       // Index 0
       IF "HMI_Interface_Overview".homeCodition[8].pageIndex = 0 THEN
           "HMI_Interface_Overview".homeCodition[8].emOverviewTitle := WSTRING#'Home Condition 0';
           "HMI_Interface_Overview".homeCodition[8].emOverviewCmName[0] := WSTRING#'Thickness Z-Axis';
           "HMI_Interface_Overview".homeCodition[8].emOverviewCmName[1] := WSTRING#'Hipot & Thickness Servo Press';
           "HMI_Interface_Overview".homeCodition[8].emOverviewCmName[2] := WSTRING#'Hipot Tab Contactor Left';
           "HMI_Interface_Overview".homeCodition[8].emOverviewCmName[3] := WSTRING#'Hipot Tab Contactor Right';
           "HMI_Interface_Overview".homeCodition[8].emOverviewCmName[4] := WSTRING#'Hipot Tab Contactor';
           "HMI_Interface_Overview".homeCodition[8].emOverviewCmName[5] := WSTRING#'Hipot & Thickness Stage Lift Front';
           "HMI_Interface_Overview".homeCodition[8].emOverviewCmName[6] := WSTRING#'Hipot & Thickness Stage Lift Rear';
           "HMI_Interface_Overview".homeCodition[8].emOverviewCmName[7] := WSTRING#'Hipot & Thickness JR Detect';
           "HMI_Interface_Overview".homeCodition[8].emOverviewCmName[8] := WSTRING#'Spare';
           "HMI_Interface_Overview".homeCodition[8].emOverviewCmName[9] := WSTRING#'Spare';
           "HMI_Interface_Overview".homeCodition[8].emOverviewCmName[10] := WSTRING#'Spare';
           "HMI_Interface_Overview".homeCodition[8].emOverviewCmName[11] := WSTRING#'Spare';
           "HMI_Interface_Overview".homeCodition[8].emOverviewCmName[12] := WSTRING#'Spare';
           "HMI_Interface_Overview".homeCodition[8].emOverviewCmName[13] := WSTRING#'Spare';
           "HMI_Interface_Overview".homeCodition[8].emOverviewCmPositionName[0] := WSTRING#'Wait Position';
           "HMI_Interface_Overview".homeCodition[8].emOverviewCmPositionName[1] := WSTRING#'Home Position';
           "HMI_Interface_Overview".homeCodition[8].emOverviewCmPositionName[2] := WSTRING#'Open';
           "HMI_Interface_Overview".homeCodition[8].emOverviewCmPositionName[3] := WSTRING#'Open';
           "HMI_Interface_Overview".homeCodition[8].emOverviewCmPositionName[4] := WSTRING#'Backward';
           "HMI_Interface_Overview".homeCodition[8].emOverviewCmPositionName[5] := WSTRING#'Down';
           "HMI_Interface_Overview".homeCodition[8].emOverviewCmPositionName[6] := WSTRING#'Down';
           "HMI_Interface_Overview".homeCodition[8].emOverviewCmPositionName[7] := WSTRING#'Not Detect';
           "HMI_Interface_Overview".homeCodition[8].emOverviewCmPositionName[8] := WSTRING#'Spare';
           "HMI_Interface_Overview".homeCodition[8].emOverviewCmPositionName[9] := WSTRING#'Spare';
           "HMI_Interface_Overview".homeCodition[8].emOverviewCmPositionName[10] := WSTRING#'Spare';
           "HMI_Interface_Overview".homeCodition[8].emOverviewCmPositionName[11] := WSTRING#'Spare';
           "HMI_Interface_Overview".homeCodition[8].emOverviewCmPositionName[12] := WSTRING#'Spare';
           "HMI_Interface_Overview".homeCodition[8].emOverviewCmPositionName[13] := WSTRING#'Spare';
           IF NOT #statLampControl THEN
               "HMI_Interface_Overview".homeCodition[8].emOverviewHomeLampOn[0] := "Unit1.Em8.HmiInterface".cm.softcam.thicknessAxisZ.pos00_wait.inPos;
               "HMI_Interface_Overview".homeCodition[8].emOverviewHomeLampOn[1] := "Unit1.Em8.HmiInterface".cmHipotThicknessServoPress.monitoring.profinetInput."HOME-POS-REACHED";
               "HMI_Interface_Overview".homeCodition[8].emOverviewHomeLampOn[2] := "Unit1.Em8.HmiInterface".cmHipotTabContactorLeftOpenClose.monitoring.inHomePos;
               "HMI_Interface_Overview".homeCodition[8].emOverviewHomeLampOn[3] := "Unit1.Em8.HmiInterface".cmHipotTabContactorRightOpenClose.monitoring.inHomePos;
               "HMI_Interface_Overview".homeCodition[8].emOverviewHomeLampOn[4] := "Unit1.Em8.HmiInterface".cmHipotTabContactorBwdFwd.monitoring.inHomePos;
               "HMI_Interface_Overview".homeCodition[8].emOverviewHomeLampOn[5] := "Unit1.Em8.HmiInterface".cmHipotThicknessStageLiftFrontUpDown.monitoring.inWorkPos;
               "HMI_Interface_Overview".homeCodition[8].emOverviewHomeLampOn[6] := "Unit1.Em8.HmiInterface".cmHipotThicknessStageLiftRearUpDown.monitoring.inWorkPos;
               "HMI_Interface_Overview".homeCodition[8].emOverviewHomeLampOn[7] := NOT "Unit1.Em8.HmiInterface".cmHipotThicknessJRDetect.monitoring.processValue;
               "HMI_Interface_Overview".homeCodition[8].emOverviewHomeLampOn[8] := FALSE;
               "HMI_Interface_Overview".homeCodition[8].emOverviewHomeLampOn[9] := FALSE;
               "HMI_Interface_Overview".homeCodition[8].emOverviewHomeLampOn[10] := FALSE;
               "HMI_Interface_Overview".homeCodition[8].emOverviewHomeLampOn[11] := FALSE;
               "HMI_Interface_Overview".homeCodition[8].emOverviewHomeLampOn[12] := FALSE;
               "HMI_Interface_Overview".homeCodition[8].emOverviewHomeLampOn[13] := FALSE;
           END_IF;
       END_IF;

       // Index 1
       IF "HMI_Interface_Overview".homeCodition[8].pageIndex = 1 THEN
           "HMI_Interface_Overview".homeCodition[8].emOverviewTitle := WSTRING#'Home Condition 1';
           "HMI_Interface_Overview".homeCodition[8].emOverviewCmName[0] := WSTRING#'Thickness Z-Axis';
           "HMI_Interface_Overview".homeCodition[8].emOverviewCmName[1] := WSTRING#'Hipot & Thickness Servo Press';
           "HMI_Interface_Overview".homeCodition[8].emOverviewCmName[2] := WSTRING#'Hipot Tab Contactor Left';
           "HMI_Interface_Overview".homeCodition[8].emOverviewCmName[3] := WSTRING#'Hipot Tab Contactor Right';
           "HMI_Interface_Overview".homeCodition[8].emOverviewCmName[4] := WSTRING#'Hipot Tab Contactor';
           "HMI_Interface_Overview".homeCodition[8].emOverviewCmName[5] := WSTRING#'Hipot & Thickness Stage Lift Front';
           "HMI_Interface_Overview".homeCodition[8].emOverviewCmName[6] := WSTRING#'Hipot & Thickness Stage Lift Rear';
           "HMI_Interface_Overview".homeCodition[8].emOverviewCmName[7] := WSTRING#'Hipot & Thickness JR Detect';
           "HMI_Interface_Overview".homeCodition[8].emOverviewCmName[8] := WSTRING#'Spare';
           "HMI_Interface_Overview".homeCodition[8].emOverviewCmName[9] := WSTRING#'Spare';
           "HMI_Interface_Overview".homeCodition[8].emOverviewCmName[10] := WSTRING#'Spare';
           "HMI_Interface_Overview".homeCodition[8].emOverviewCmName[11] := WSTRING#'Spare';
           "HMI_Interface_Overview".homeCodition[8].emOverviewCmName[12] := WSTRING#'Spare';
           "HMI_Interface_Overview".homeCodition[8].emOverviewCmName[13] := WSTRING#'Spare';
           "HMI_Interface_Overview".homeCodition[8].emOverviewCmPositionName[0] := WSTRING#'Wait Position';
           "HMI_Interface_Overview".homeCodition[8].emOverviewCmPositionName[1] := WSTRING#'Home Position';
           "HMI_Interface_Overview".homeCodition[8].emOverviewCmPositionName[2] := WSTRING#'Open';
           "HMI_Interface_Overview".homeCodition[8].emOverviewCmPositionName[3] := WSTRING#'Open';
           "HMI_Interface_Overview".homeCodition[8].emOverviewCmPositionName[4] := WSTRING#'Backward';
           "HMI_Interface_Overview".homeCodition[8].emOverviewCmPositionName[5] := WSTRING#'Down';
           "HMI_Interface_Overview".homeCodition[8].emOverviewCmPositionName[6] := WSTRING#'Down';
           "HMI_Interface_Overview".homeCodition[8].emOverviewCmPositionName[7] := WSTRING#'Detect';
           "HMI_Interface_Overview".homeCodition[8].emOverviewCmPositionName[8] := WSTRING#'Spare';
           "HMI_Interface_Overview".homeCodition[8].emOverviewCmPositionName[9] := WSTRING#'Spare';
           "HMI_Interface_Overview".homeCodition[8].emOverviewCmPositionName[10] := WSTRING#'Spare';
           "HMI_Interface_Overview".homeCodition[8].emOverviewCmPositionName[11] := WSTRING#'Spare';
           "HMI_Interface_Overview".homeCodition[8].emOverviewCmPositionName[12] := WSTRING#'Spare';
           "HMI_Interface_Overview".homeCodition[8].emOverviewCmPositionName[13] := WSTRING#'Spare';
           IF NOT #statLampControl THEN
               "HMI_Interface_Overview".homeCodition[8].emOverviewHomeLampOn[0] := "Unit1.Em8.HmiInterface".cm.softcam.thicknessAxisZ.pos00_wait.inPos;
               "HMI_Interface_Overview".homeCodition[8].emOverviewHomeLampOn[1] := "Unit1.Em8.HmiInterface".cmHipotThicknessServoPress.monitoring.profinetInput."HOME-POS-REACHED";
               "HMI_Interface_Overview".homeCodition[8].emOverviewHomeLampOn[2] := "Unit1.Em8.HmiInterface".cmHipotTabContactorLeftOpenClose.monitoring.inHomePos;
               "HMI_Interface_Overview".homeCodition[8].emOverviewHomeLampOn[3] := "Unit1.Em8.HmiInterface".cmHipotTabContactorRightOpenClose.monitoring.inHomePos;
               "HMI_Interface_Overview".homeCodition[8].emOverviewHomeLampOn[4] := "Unit1.Em8.HmiInterface".cmHipotTabContactorBwdFwd.monitoring.inHomePos;
               "HMI_Interface_Overview".homeCodition[8].emOverviewHomeLampOn[5] := "Unit1.Em8.HmiInterface".cmHipotThicknessStageLiftFrontUpDown.monitoring.inWorkPos;
               "HMI_Interface_Overview".homeCodition[8].emOverviewHomeLampOn[6] := "Unit1.Em8.HmiInterface".cmHipotThicknessStageLiftRearUpDown.monitoring.inWorkPos;
               "HMI_Interface_Overview".homeCodition[8].emOverviewHomeLampOn[7] := "Unit1.Em8.HmiInterface".cmHipotThicknessJRDetect.monitoring.processValue;
               "HMI_Interface_Overview".homeCodition[8].emOverviewHomeLampOn[8] := FALSE;
               "HMI_Interface_Overview".homeCodition[8].emOverviewHomeLampOn[9] := FALSE;
               "HMI_Interface_Overview".homeCodition[8].emOverviewHomeLampOn[10] := FALSE;
               "HMI_Interface_Overview".homeCodition[8].emOverviewHomeLampOn[11] := FALSE;
               "HMI_Interface_Overview".homeCodition[8].emOverviewHomeLampOn[12] := FALSE;
               "HMI_Interface_Overview".homeCodition[8].emOverviewHomeLampOn[13] := FALSE;
           END_IF;
       END_IF;

   END_REGION
END_REGION

REGION Network 39 (SCL): Em 9 Page Index Mapping
   REGION Page Index

       // Index 0
       IF "HMI_Interface_Overview".homeCodition[9].pageIndex = 0 THEN
           "HMI_Interface_Overview".homeCodition[9].emOverviewTitle := WSTRING#'Home Condition 0';
           "HMI_Interface_Overview".homeCodition[9].emOverviewCmName[0] := WSTRING#'Vision Stage Lift';
           "HMI_Interface_Overview".homeCodition[9].emOverviewCmName[1] := WSTRING#'Vision Light';
           "HMI_Interface_Overview".homeCodition[9].emOverviewCmName[2] := WSTRING#'Vision JR Detect';
           "HMI_Interface_Overview".homeCodition[9].emOverviewCmName[3] := WSTRING#'Spare';
           "HMI_Interface_Overview".homeCodition[9].emOverviewCmName[4] := WSTRING#'Spare';
           "HMI_Interface_Overview".homeCodition[9].emOverviewCmName[5] := WSTRING#'Spare';
           "HMI_Interface_Overview".homeCodition[9].emOverviewCmName[6] := WSTRING#'Spare';
           "HMI_Interface_Overview".homeCodition[9].emOverviewCmName[7] := WSTRING#'Spare';
           "HMI_Interface_Overview".homeCodition[9].emOverviewCmName[8] := WSTRING#'Spare';
           "HMI_Interface_Overview".homeCodition[9].emOverviewCmName[9] := WSTRING#'Spare';
           "HMI_Interface_Overview".homeCodition[9].emOverviewCmName[10] := WSTRING#'Spare';
           "HMI_Interface_Overview".homeCodition[9].emOverviewCmName[11] := WSTRING#'Spare';
           "HMI_Interface_Overview".homeCodition[9].emOverviewCmName[12] := WSTRING#'Spare';
           "HMI_Interface_Overview".homeCodition[9].emOverviewCmName[13] := WSTRING#'Spare';
           "HMI_Interface_Overview".homeCodition[9].emOverviewCmPositionName[0] := WSTRING#'Down';
           "HMI_Interface_Overview".homeCodition[9].emOverviewCmPositionName[1] := WSTRING#'Up';
           "HMI_Interface_Overview".homeCodition[9].emOverviewCmPositionName[2] := WSTRING#'Not Detect';
           "HMI_Interface_Overview".homeCodition[9].emOverviewCmPositionName[3] := WSTRING#'Spare';
           "HMI_Interface_Overview".homeCodition[9].emOverviewCmPositionName[4] := WSTRING#'Spare';
           "HMI_Interface_Overview".homeCodition[9].emOverviewCmPositionName[5] := WSTRING#'Spare';
           "HMI_Interface_Overview".homeCodition[9].emOverviewCmPositionName[6] := WSTRING#'Spare';
           "HMI_Interface_Overview".homeCodition[9].emOverviewCmPositionName[7] := WSTRING#'Spare';
           "HMI_Interface_Overview".homeCodition[9].emOverviewCmPositionName[8] := WSTRING#'Spare';
           "HMI_Interface_Overview".homeCodition[9].emOverviewCmPositionName[9] := WSTRING#'Spare';
           "HMI_Interface_Overview".homeCodition[9].emOverviewCmPositionName[10] := WSTRING#'Spare';
           "HMI_Interface_Overview".homeCodition[9].emOverviewCmPositionName[11] := WSTRING#'Spare';
           "HMI_Interface_Overview".homeCodition[9].emOverviewCmPositionName[12] := WSTRING#'Spare';
           "HMI_Interface_Overview".homeCodition[9].emOverviewCmPositionName[13] := WSTRING#'Spare';
           IF NOT #statLampControl THEN
               "HMI_Interface_Overview".homeCodition[9].emOverviewHomeLampOn[0] := "Unit1.Em9.HmiInterface".cmVisionStageLiftUpDown.monitoring.inWorkPos;
               "HMI_Interface_Overview".homeCodition[9].emOverviewHomeLampOn[1] := "Unit1.Em9.HmiInterface".cmVisionLightUpDown.monitoring.inHomePos;
               "HMI_Interface_Overview".homeCodition[9].emOverviewHomeLampOn[2] := NOT "Unit1.Em9.HmiInterface".cmVisionJRDetect.monitoring.processValue;
               "HMI_Interface_Overview".homeCodition[9].emOverviewHomeLampOn[3] := FALSE;
               "HMI_Interface_Overview".homeCodition[9].emOverviewHomeLampOn[4] := FALSE;
               "HMI_Interface_Overview".homeCodition[9].emOverviewHomeLampOn[5] := FALSE;
               "HMI_Interface_Overview".homeCodition[9].emOverviewHomeLampOn[6] := FALSE;
               "HMI_Interface_Overview".homeCodition[9].emOverviewHomeLampOn[7] := FALSE;
               "HMI_Interface_Overview".homeCodition[9].emOverviewHomeLampOn[8] := FALSE;
               "HMI_Interface_Overview".homeCodition[9].emOverviewHomeLampOn[9] := FALSE;
               "HMI_Interface_Overview".homeCodition[9].emOverviewHomeLampOn[10] := FALSE;
               "HMI_Interface_Overview".homeCodition[9].emOverviewHomeLampOn[11] := FALSE;
               "HMI_Interface_Overview".homeCodition[9].emOverviewHomeLampOn[12] := FALSE;
               "HMI_Interface_Overview".homeCodition[9].emOverviewHomeLampOn[13] := FALSE;
           END_IF;
       END_IF;

       // Index 1
       IF "HMI_Interface_Overview".homeCodition[9].pageIndex = 1 THEN
           "HMI_Interface_Overview".homeCodition[9].emOverviewTitle := WSTRING#'Home Condition 1';
           "HMI_Interface_Overview".homeCodition[9].emOverviewCmName[0] := WSTRING#'Vision Stage Lift';
           "HMI_Interface_Overview".homeCodition[9].emOverviewCmName[1] := WSTRING#'Vision Light';
           "HMI_Interface_Overview".homeCodition[9].emOverviewCmName[2] := WSTRING#'Vision JR Detect';
           "HMI_Interface_Overview".homeCodition[9].emOverviewCmName[3] := WSTRING#'Spare';
           "HMI_Interface_Overview".homeCodition[9].emOverviewCmName[4] := WSTRING#'Spare';
           "HMI_Interface_Overview".homeCodition[9].emOverviewCmName[5] := WSTRING#'Spare';
           "HMI_Interface_Overview".homeCodition[9].emOverviewCmName[6] := WSTRING#'Spare';
           "HMI_Interface_Overview".homeCodition[9].emOverviewCmName[7] := WSTRING#'Spare';
           "HMI_Interface_Overview".homeCodition[9].emOverviewCmName[8] := WSTRING#'Spare';
           "HMI_Interface_Overview".homeCodition[9].emOverviewCmName[9] := WSTRING#'Spare';
           "HMI_Interface_Overview".homeCodition[9].emOverviewCmName[10] := WSTRING#'Spare';
           "HMI_Interface_Overview".homeCodition[9].emOverviewCmName[11] := WSTRING#'Spare';
           "HMI_Interface_Overview".homeCodition[9].emOverviewCmName[12] := WSTRING#'Spare';
           "HMI_Interface_Overview".homeCodition[9].emOverviewCmName[13] := WSTRING#'Spare';
           "HMI_Interface_Overview".homeCodition[9].emOverviewCmPositionName[0] := WSTRING#'Down';
           "HMI_Interface_Overview".homeCodition[9].emOverviewCmPositionName[1] := WSTRING#'Up';
           "HMI_Interface_Overview".homeCodition[9].emOverviewCmPositionName[2] := WSTRING#'Detect';
           "HMI_Interface_Overview".homeCodition[9].emOverviewCmPositionName[3] := WSTRING#'Spare';
           "HMI_Interface_Overview".homeCodition[9].emOverviewCmPositionName[4] := WSTRING#'Spare';
           "HMI_Interface_Overview".homeCodition[9].emOverviewCmPositionName[5] := WSTRING#'Spare';
           "HMI_Interface_Overview".homeCodition[9].emOverviewCmPositionName[6] := WSTRING#'Spare';
           "HMI_Interface_Overview".homeCodition[9].emOverviewCmPositionName[7] := WSTRING#'Spare';
           "HMI_Interface_Overview".homeCodition[9].emOverviewCmPositionName[8] := WSTRING#'Spare';
           "HMI_Interface_Overview".homeCodition[9].emOverviewCmPositionName[9] := WSTRING#'Spare';
           "HMI_Interface_Overview".homeCodition[9].emOverviewCmPositionName[10] := WSTRING#'Spare';
           "HMI_Interface_Overview".homeCodition[9].emOverviewCmPositionName[11] := WSTRING#'Spare';
           "HMI_Interface_Overview".homeCodition[9].emOverviewCmPositionName[12] := WSTRING#'Spare';
           "HMI_Interface_Overview".homeCodition[9].emOverviewCmPositionName[13] := WSTRING#'Spare';
           IF NOT #statLampControl THEN
               "HMI_Interface_Overview".homeCodition[9].emOverviewHomeLampOn[0] := "Unit1.Em9.HmiInterface".cmVisionStageLiftUpDown.monitoring.inWorkPos;
               "HMI_Interface_Overview".homeCodition[9].emOverviewHomeLampOn[1] := "Unit1.Em9.HmiInterface".cmVisionLightUpDown.monitoring.inHomePos;
               "HMI_Interface_Overview".homeCodition[9].emOverviewHomeLampOn[2] := "Unit1.Em9.HmiInterface".cmVisionJRDetect.monitoring.processValue;
               "HMI_Interface_Overview".homeCodition[9].emOverviewHomeLampOn[3] := FALSE;
               "HMI_Interface_Overview".homeCodition[9].emOverviewHomeLampOn[4] := FALSE;
               "HMI_Interface_Overview".homeCodition[9].emOverviewHomeLampOn[5] := FALSE;
               "HMI_Interface_Overview".homeCodition[9].emOverviewHomeLampOn[6] := FALSE;
               "HMI_Interface_Overview".homeCodition[9].emOverviewHomeLampOn[7] := FALSE;
               "HMI_Interface_Overview".homeCodition[9].emOverviewHomeLampOn[8] := FALSE;
               "HMI_Interface_Overview".homeCodition[9].emOverviewHomeLampOn[9] := FALSE;
               "HMI_Interface_Overview".homeCodition[9].emOverviewHomeLampOn[10] := FALSE;
               "HMI_Interface_Overview".homeCodition[9].emOverviewHomeLampOn[11] := FALSE;
               "HMI_Interface_Overview".homeCodition[9].emOverviewHomeLampOn[12] := FALSE;
               "HMI_Interface_Overview".homeCodition[9].emOverviewHomeLampOn[13] := FALSE;
           END_IF;
       END_IF;

   END_REGION
END_REGION

REGION Network 40 (SCL): Em 10 Page Index Mapping
   REGION Page Index

       // Index 0
       IF "HMI_Interface_Overview".homeCodition[10].pageIndex = 0 THEN
           "HMI_Interface_Overview".homeCodition[10].emOverviewTitle := WSTRING#'Home Condition 0';
           "HMI_Interface_Overview".homeCodition[10].emOverviewCmName[0] := WSTRING#'Laser Mark Stage Lift';
           "HMI_Interface_Overview".homeCodition[10].emOverviewCmName[1] := WSTRING#'Laser Mark Cover';
           "HMI_Interface_Overview".homeCodition[10].emOverviewCmName[2] := WSTRING#'Laser Mark JR Detect';
           "HMI_Interface_Overview".homeCodition[10].emOverviewCmName[3] := WSTRING#'Spare';
           "HMI_Interface_Overview".homeCodition[10].emOverviewCmName[4] := WSTRING#'Spare';
           "HMI_Interface_Overview".homeCodition[10].emOverviewCmName[5] := WSTRING#'Spare';
           "HMI_Interface_Overview".homeCodition[10].emOverviewCmName[6] := WSTRING#'Spare';
           "HMI_Interface_Overview".homeCodition[10].emOverviewCmName[7] := WSTRING#'Spare';
           "HMI_Interface_Overview".homeCodition[10].emOverviewCmName[8] := WSTRING#'Spare';
           "HMI_Interface_Overview".homeCodition[10].emOverviewCmName[9] := WSTRING#'Spare';
           "HMI_Interface_Overview".homeCodition[10].emOverviewCmName[10] := WSTRING#'Spare';
           "HMI_Interface_Overview".homeCodition[10].emOverviewCmName[11] := WSTRING#'Spare';
           "HMI_Interface_Overview".homeCodition[10].emOverviewCmName[12] := WSTRING#'Spare';
           "HMI_Interface_Overview".homeCodition[10].emOverviewCmName[13] := WSTRING#'Spare';
           "HMI_Interface_Overview".homeCodition[10].emOverviewCmPositionName[0] := WSTRING#'Down';
           "HMI_Interface_Overview".homeCodition[10].emOverviewCmPositionName[1] := WSTRING#'Up';
           "HMI_Interface_Overview".homeCodition[10].emOverviewCmPositionName[2] := WSTRING#'Not Detect';
           "HMI_Interface_Overview".homeCodition[10].emOverviewCmPositionName[3] := WSTRING#'Spare';
           "HMI_Interface_Overview".homeCodition[10].emOverviewCmPositionName[4] := WSTRING#'Spare';
           "HMI_Interface_Overview".homeCodition[10].emOverviewCmPositionName[5] := WSTRING#'Spare';
           "HMI_Interface_Overview".homeCodition[10].emOverviewCmPositionName[6] := WSTRING#'Spare';
           "HMI_Interface_Overview".homeCodition[10].emOverviewCmPositionName[7] := WSTRING#'Spare';
           "HMI_Interface_Overview".homeCodition[10].emOverviewCmPositionName[8] := WSTRING#'Spare';
           "HMI_Interface_Overview".homeCodition[10].emOverviewCmPositionName[9] := WSTRING#'Spare';
           "HMI_Interface_Overview".homeCodition[10].emOverviewCmPositionName[10] := WSTRING#'Spare';
           "HMI_Interface_Overview".homeCodition[10].emOverviewCmPositionName[11] := WSTRING#'Spare';
           "HMI_Interface_Overview".homeCodition[10].emOverviewCmPositionName[12] := WSTRING#'Spare';
           "HMI_Interface_Overview".homeCodition[10].emOverviewCmPositionName[13] := WSTRING#'Spare';
           IF NOT #statLampControl THEN
               "HMI_Interface_Overview".homeCodition[10].emOverviewHomeLampOn[0] := "Unit1.Em10.HmiInterface".cmLaserMarkStageLiftUpDown.monitoring.inWorkPos;
               "HMI_Interface_Overview".homeCodition[10].emOverviewHomeLampOn[1] := "Unit1.Em10.HmiInterface".cmLaserMarkCoverUpDown.monitoring.inHomePos;
               "HMI_Interface_Overview".homeCodition[10].emOverviewHomeLampOn[2] := NOT "Unit1.Em10.HmiInterface".cmLaserMarkJRDetect.monitoring.processValue;
               "HMI_Interface_Overview".homeCodition[10].emOverviewHomeLampOn[3] := FALSE;
               "HMI_Interface_Overview".homeCodition[10].emOverviewHomeLampOn[4] := FALSE;
               "HMI_Interface_Overview".homeCodition[10].emOverviewHomeLampOn[5] := FALSE;
               "HMI_Interface_Overview".homeCodition[10].emOverviewHomeLampOn[6] := FALSE;
               "HMI_Interface_Overview".homeCodition[10].emOverviewHomeLampOn[7] := FALSE;
               "HMI_Interface_Overview".homeCodition[10].emOverviewHomeLampOn[8] := FALSE;
               "HMI_Interface_Overview".homeCodition[10].emOverviewHomeLampOn[9] := FALSE;
               "HMI_Interface_Overview".homeCodition[10].emOverviewHomeLampOn[10] := FALSE;
               "HMI_Interface_Overview".homeCodition[10].emOverviewHomeLampOn[11] := FALSE;
               "HMI_Interface_Overview".homeCodition[10].emOverviewHomeLampOn[12] := FALSE;
               "HMI_Interface_Overview".homeCodition[10].emOverviewHomeLampOn[13] := FALSE;
           END_IF;
       END_IF;

       // Index 1
       IF "HMI_Interface_Overview".homeCodition[10].pageIndex = 1 THEN
           "HMI_Interface_Overview".homeCodition[10].emOverviewTitle := WSTRING#'Home Condition 1';
           "HMI_Interface_Overview".homeCodition[10].emOverviewCmName[0] := WSTRING#'Laser Mark Stage Lift';
           "HMI_Interface_Overview".homeCodition[10].emOverviewCmName[1] := WSTRING#'Laser Mark Cover';
           "HMI_Interface_Overview".homeCodition[10].emOverviewCmName[2] := WSTRING#'Laser Mark JR Detect';
           "HMI_Interface_Overview".homeCodition[10].emOverviewCmName[3] := WSTRING#'Spare';
           "HMI_Interface_Overview".homeCodition[10].emOverviewCmName[4] := WSTRING#'Spare';
           "HMI_Interface_Overview".homeCodition[10].emOverviewCmName[5] := WSTRING#'Spare';
           "HMI_Interface_Overview".homeCodition[10].emOverviewCmName[6] := WSTRING#'Spare';
           "HMI_Interface_Overview".homeCodition[10].emOverviewCmName[7] := WSTRING#'Spare';
           "HMI_Interface_Overview".homeCodition[10].emOverviewCmName[8] := WSTRING#'Spare';
           "HMI_Interface_Overview".homeCodition[10].emOverviewCmName[9] := WSTRING#'Spare';
           "HMI_Interface_Overview".homeCodition[10].emOverviewCmName[10] := WSTRING#'Spare';
           "HMI_Interface_Overview".homeCodition[10].emOverviewCmName[11] := WSTRING#'Spare';
           "HMI_Interface_Overview".homeCodition[10].emOverviewCmName[12] := WSTRING#'Spare';
           "HMI_Interface_Overview".homeCodition[10].emOverviewCmName[13] := WSTRING#'Spare';
           "HMI_Interface_Overview".homeCodition[10].emOverviewCmPositionName[0] := WSTRING#'Down';
           "HMI_Interface_Overview".homeCodition[10].emOverviewCmPositionName[1] := WSTRING#'Up';
           "HMI_Interface_Overview".homeCodition[10].emOverviewCmPositionName[2] := WSTRING#'Detect';
           "HMI_Interface_Overview".homeCodition[10].emOverviewCmPositionName[3] := WSTRING#'Spare';
           "HMI_Interface_Overview".homeCodition[10].emOverviewCmPositionName[4] := WSTRING#'Spare';
           "HMI_Interface_Overview".homeCodition[10].emOverviewCmPositionName[5] := WSTRING#'Spare';
           "HMI_Interface_Overview".homeCodition[10].emOverviewCmPositionName[6] := WSTRING#'Spare';
           "HMI_Interface_Overview".homeCodition[10].emOverviewCmPositionName[7] := WSTRING#'Spare';
           "HMI_Interface_Overview".homeCodition[10].emOverviewCmPositionName[8] := WSTRING#'Spare';
           "HMI_Interface_Overview".homeCodition[10].emOverviewCmPositionName[9] := WSTRING#'Spare';
           "HMI_Interface_Overview".homeCodition[10].emOverviewCmPositionName[10] := WSTRING#'Spare';
           "HMI_Interface_Overview".homeCodition[10].emOverviewCmPositionName[11] := WSTRING#'Spare';
           "HMI_Interface_Overview".homeCodition[10].emOverviewCmPositionName[12] := WSTRING#'Spare';
           "HMI_Interface_Overview".homeCodition[10].emOverviewCmPositionName[13] := WSTRING#'Spare';
           IF NOT #statLampControl THEN
               "HMI_Interface_Overview".homeCodition[10].emOverviewHomeLampOn[0] := "Unit1.Em10.HmiInterface".cmLaserMarkStageLiftUpDown.monitoring.inWorkPos;
               "HMI_Interface_Overview".homeCodition[10].emOverviewHomeLampOn[1] := "Unit1.Em10.HmiInterface".cmLaserMarkCoverUpDown.monitoring.inHomePos;
               "HMI_Interface_Overview".homeCodition[10].emOverviewHomeLampOn[2] := "Unit1.Em10.HmiInterface".cmLaserMarkJRDetect.monitoring.processValue;
               "HMI_Interface_Overview".homeCodition[10].emOverviewHomeLampOn[3] := FALSE;
               "HMI_Interface_Overview".homeCodition[10].emOverviewHomeLampOn[4] := FALSE;
               "HMI_Interface_Overview".homeCodition[10].emOverviewHomeLampOn[5] := FALSE;
               "HMI_Interface_Overview".homeCodition[10].emOverviewHomeLampOn[6] := FALSE;
               "HMI_Interface_Overview".homeCodition[10].emOverviewHomeLampOn[7] := FALSE;
               "HMI_Interface_Overview".homeCodition[10].emOverviewHomeLampOn[8] := FALSE;
               "HMI_Interface_Overview".homeCodition[10].emOverviewHomeLampOn[9] := FALSE;
               "HMI_Interface_Overview".homeCodition[10].emOverviewHomeLampOn[10] := FALSE;
               "HMI_Interface_Overview".homeCodition[10].emOverviewHomeLampOn[11] := FALSE;
               "HMI_Interface_Overview".homeCodition[10].emOverviewHomeLampOn[12] := FALSE;
               "HMI_Interface_Overview".homeCodition[10].emOverviewHomeLampOn[13] := FALSE;
           END_IF;
       END_IF;

   END_REGION
END_REGION

REGION Network 41 (SCL): Em 12 Page Index Mapping
   REGION Page Index

       // Index 0
       IF "HMI_Interface_Overview".homeCodition[12].pageIndex = 0 THEN
           "HMI_Interface_Overview".homeCodition[12].emOverviewTitle := WSTRING#'Home Condition 0';
           "HMI_Interface_Overview".homeCodition[12].emOverviewCmName[0] := WSTRING#'Stack NG Box Loading';
           "HMI_Interface_Overview".homeCodition[12].emOverviewCmName[1] := WSTRING#'Stack NG Box Unit Mover';
           "HMI_Interface_Overview".homeCodition[12].emOverviewCmName[2] := WSTRING#'Stack NG Box Clamp Left ';
           "HMI_Interface_Overview".homeCodition[12].emOverviewCmName[3] := WSTRING#'Stack NG Box Clamp Right';
           "HMI_Interface_Overview".homeCodition[12].emOverviewCmName[4] := WSTRING#'Stack NG Box Clamp Mover';
           "HMI_Interface_Overview".homeCodition[12].emOverviewCmName[5] := WSTRING#'Spare';
           "HMI_Interface_Overview".homeCodition[12].emOverviewCmName[6] := WSTRING#'Spare';
           "HMI_Interface_Overview".homeCodition[12].emOverviewCmName[7] := WSTRING#'Spare';
           "HMI_Interface_Overview".homeCodition[12].emOverviewCmName[8] := WSTRING#'Spare';
           "HMI_Interface_Overview".homeCodition[12].emOverviewCmName[9] := WSTRING#'Spare';
           "HMI_Interface_Overview".homeCodition[12].emOverviewCmName[10] := WSTRING#'Spare';
           "HMI_Interface_Overview".homeCodition[12].emOverviewCmName[11] := WSTRING#'Spare';
           "HMI_Interface_Overview".homeCodition[12].emOverviewCmName[12] := WSTRING#'Spare';
           "HMI_Interface_Overview".homeCodition[12].emOverviewCmName[13] := WSTRING#'Spare';
           "HMI_Interface_Overview".homeCodition[12].emOverviewCmPositionName[0] := WSTRING#'Up';
           "HMI_Interface_Overview".homeCodition[12].emOverviewCmPositionName[1] := WSTRING#'Forward';
           "HMI_Interface_Overview".homeCodition[12].emOverviewCmPositionName[2] := WSTRING#'Open';
           "HMI_Interface_Overview".homeCodition[12].emOverviewCmPositionName[3] := WSTRING#'Open';
           "HMI_Interface_Overview".homeCodition[12].emOverviewCmPositionName[4] := WSTRING#'Open';
           "HMI_Interface_Overview".homeCodition[12].emOverviewCmPositionName[5] := WSTRING#'Spare';
           "HMI_Interface_Overview".homeCodition[12].emOverviewCmPositionName[6] := WSTRING#'Spare';
           "HMI_Interface_Overview".homeCodition[12].emOverviewCmPositionName[7] := WSTRING#'Spare';
           "HMI_Interface_Overview".homeCodition[12].emOverviewCmPositionName[8] := WSTRING#'Spare';
           "HMI_Interface_Overview".homeCodition[12].emOverviewCmPositionName[9] := WSTRING#'Spare';
           "HMI_Interface_Overview".homeCodition[12].emOverviewCmPositionName[10] := WSTRING#'Spare';
           "HMI_Interface_Overview".homeCodition[12].emOverviewCmPositionName[11] := WSTRING#'Spare';
           "HMI_Interface_Overview".homeCodition[12].emOverviewCmPositionName[12] := WSTRING#'Spare';
           "HMI_Interface_Overview".homeCodition[12].emOverviewCmPositionName[13] := WSTRING#'Spare';
           IF NOT #statLampControl THEN
               "HMI_Interface_Overview".homeCodition[12].emOverviewHomeLampOn[0] := "Unit1.Em12.HmiInterface".cmStackNgBoxLoadingUpDown.monitoring.inHomePos;
               "HMI_Interface_Overview".homeCodition[12].emOverviewHomeLampOn[1] := "Unit1.Em12.HmiInterface".cmStackNgBoxUnitMoverBwdFwd.monitoring.inWorkPos;
               "HMI_Interface_Overview".homeCodition[12].emOverviewHomeLampOn[2] := "Unit1.Em12.HmiInterface".cmStackNgBoxClampLeftOpenClose.monitoring.inHomePos;
               "HMI_Interface_Overview".homeCodition[12].emOverviewHomeLampOn[3] := "Unit1.Em12.HmiInterface".cmStackNgBoxClampRightOpenClose.monitoring.inHomePos;
               "HMI_Interface_Overview".homeCodition[12].emOverviewHomeLampOn[4] := "Unit1.Em12.HmiInterface".cmStackNgBoxClampMoverOpenClose.monitoring.inHomePos;
               "HMI_Interface_Overview".homeCodition[12].emOverviewHomeLampOn[5] := FALSE;
               "HMI_Interface_Overview".homeCodition[12].emOverviewHomeLampOn[6] := FALSE;
               "HMI_Interface_Overview".homeCodition[12].emOverviewHomeLampOn[7] := FALSE;
               "HMI_Interface_Overview".homeCodition[12].emOverviewHomeLampOn[8] := FALSE;
               "HMI_Interface_Overview".homeCodition[12].emOverviewHomeLampOn[9] := FALSE;
               "HMI_Interface_Overview".homeCodition[12].emOverviewHomeLampOn[10] := FALSE;
               "HMI_Interface_Overview".homeCodition[12].emOverviewHomeLampOn[11] := FALSE;
               "HMI_Interface_Overview".homeCodition[12].emOverviewHomeLampOn[12] := FALSE;
               "HMI_Interface_Overview".homeCodition[12].emOverviewHomeLampOn[13] := FALSE;
           END_IF;
       END_IF;

       // Index 1
       IF "HMI_Interface_Overview".homeCodition[12].pageIndex = 1 THEN
           "HMI_Interface_Overview".homeCodition[12].emOverviewTitle := WSTRING#'Home Condition 1';
           "HMI_Interface_Overview".homeCodition[12].emOverviewCmName[0] := WSTRING#'Stack NG Box Loading';
           "HMI_Interface_Overview".homeCodition[12].emOverviewCmName[1] := WSTRING#'Stack NG Box Unit Mover';
           "HMI_Interface_Overview".homeCodition[12].emOverviewCmName[2] := WSTRING#'Stack NG Box Clamp Left ';
           "HMI_Interface_Overview".homeCodition[12].emOverviewCmName[3] := WSTRING#'Stack NG Box Clamp Right';
           "HMI_Interface_Overview".homeCodition[12].emOverviewCmName[4] := WSTRING#'Stack NG Box Clamp Mover';
           "HMI_Interface_Overview".homeCodition[12].emOverviewCmName[5] := WSTRING#'Spare';
           "HMI_Interface_Overview".homeCodition[12].emOverviewCmName[6] := WSTRING#'Spare';
           "HMI_Interface_Overview".homeCodition[12].emOverviewCmName[7] := WSTRING#'Spare';
           "HMI_Interface_Overview".homeCodition[12].emOverviewCmName[8] := WSTRING#'Spare';
           "HMI_Interface_Overview".homeCodition[12].emOverviewCmName[9] := WSTRING#'Spare';
           "HMI_Interface_Overview".homeCodition[12].emOverviewCmName[10] := WSTRING#'Spare';
           "HMI_Interface_Overview".homeCodition[12].emOverviewCmName[11] := WSTRING#'Spare';
           "HMI_Interface_Overview".homeCodition[12].emOverviewCmName[12] := WSTRING#'Spare';
           "HMI_Interface_Overview".homeCodition[12].emOverviewCmName[13] := WSTRING#'Spare';
           "HMI_Interface_Overview".homeCodition[12].emOverviewCmPositionName[0] := WSTRING#'Up';
           "HMI_Interface_Overview".homeCodition[12].emOverviewCmPositionName[1] := WSTRING#'Forward';
           "HMI_Interface_Overview".homeCodition[12].emOverviewCmPositionName[2] := WSTRING#'Close';
           "HMI_Interface_Overview".homeCodition[12].emOverviewCmPositionName[3] := WSTRING#'Close';
           "HMI_Interface_Overview".homeCodition[12].emOverviewCmPositionName[4] := WSTRING#'Close';
           "HMI_Interface_Overview".homeCodition[12].emOverviewCmPositionName[5] := WSTRING#'Spare';
           "HMI_Interface_Overview".homeCodition[12].emOverviewCmPositionName[6] := WSTRING#'Spare';
           "HMI_Interface_Overview".homeCodition[12].emOverviewCmPositionName[7] := WSTRING#'Spare';
           "HMI_Interface_Overview".homeCodition[12].emOverviewCmPositionName[8] := WSTRING#'Spare';
           "HMI_Interface_Overview".homeCodition[12].emOverviewCmPositionName[9] := WSTRING#'Spare';
           "HMI_Interface_Overview".homeCodition[12].emOverviewCmPositionName[10] := WSTRING#'Spare';
           "HMI_Interface_Overview".homeCodition[12].emOverviewCmPositionName[11] := WSTRING#'Spare';
           "HMI_Interface_Overview".homeCodition[12].emOverviewCmPositionName[12] := WSTRING#'Spare';
           "HMI_Interface_Overview".homeCodition[12].emOverviewCmPositionName[13] := WSTRING#'Spare';
           IF NOT #statLampControl THEN
               "HMI_Interface_Overview".homeCodition[12].emOverviewHomeLampOn[0] := "Unit1.Em12.HmiInterface".cmStackNgBoxLoadingUpDown.monitoring.inHomePos;
               "HMI_Interface_Overview".homeCodition[12].emOverviewHomeLampOn[1] := "Unit1.Em12.HmiInterface".cmStackNgBoxUnitMoverBwdFwd.monitoring.inWorkPos;
               "HMI_Interface_Overview".homeCodition[12].emOverviewHomeLampOn[2] := "Unit1.Em12.HmiInterface".cmStackNgBoxClampLeftOpenClose.monitoring.inWorkPos;
               "HMI_Interface_Overview".homeCodition[12].emOverviewHomeLampOn[3] := "Unit1.Em12.HmiInterface".cmStackNgBoxClampRightOpenClose.monitoring.inWorkPos;
               "HMI_Interface_Overview".homeCodition[12].emOverviewHomeLampOn[4] := "Unit1.Em12.HmiInterface".cmStackNgBoxClampMoverOpenClose.monitoring.inWorkPos;
               "HMI_Interface_Overview".homeCodition[12].emOverviewHomeLampOn[5] := FALSE;
               "HMI_Interface_Overview".homeCodition[12].emOverviewHomeLampOn[6] := FALSE;
               "HMI_Interface_Overview".homeCodition[12].emOverviewHomeLampOn[7] := FALSE;
               "HMI_Interface_Overview".homeCodition[12].emOverviewHomeLampOn[8] := FALSE;
               "HMI_Interface_Overview".homeCodition[12].emOverviewHomeLampOn[9] := FALSE;
               "HMI_Interface_Overview".homeCodition[12].emOverviewHomeLampOn[10] := FALSE;
               "HMI_Interface_Overview".homeCodition[12].emOverviewHomeLampOn[11] := FALSE;
               "HMI_Interface_Overview".homeCodition[12].emOverviewHomeLampOn[12] := FALSE;
               "HMI_Interface_Overview".homeCodition[12].emOverviewHomeLampOn[13] := FALSE;
           END_IF;
       END_IF;

   END_REGION
END_REGION

REGION Network 42 (SCL): Em 13 Page Index Mapping
   REGION Page Index

       // Index 0
       IF "HMI_Interface_Overview".homeCodition[13].pageIndex = 0 THEN
           "HMI_Interface_Overview".homeCodition[13].emOverviewTitle := WSTRING#'Home Condition 0';
           "HMI_Interface_Overview".homeCodition[13].emOverviewCmName[0] := WSTRING#'JR Unloading P&P X-Axis';
           "HMI_Interface_Overview".homeCodition[13].emOverviewCmName[1] := WSTRING#'JR Unloading P&P Z-Axis';
           "HMI_Interface_Overview".homeCodition[13].emOverviewCmName[2] := WSTRING#'JR Unloading P&P C-Axis';
           "HMI_Interface_Overview".homeCodition[13].emOverviewCmName[3] := WSTRING#'JR Unloading P&P Clamp';
           "HMI_Interface_Overview".homeCodition[13].emOverviewCmName[4] := WSTRING#'JR Unloading P&P JR Detect';
           "HMI_Interface_Overview".homeCodition[13].emOverviewCmName[5] := WSTRING#'Spare';
           "HMI_Interface_Overview".homeCodition[13].emOverviewCmName[6] := WSTRING#'Spare';
           "HMI_Interface_Overview".homeCodition[13].emOverviewCmName[7] := WSTRING#'Spare';
           "HMI_Interface_Overview".homeCodition[13].emOverviewCmName[8] := WSTRING#'Spare';
           "HMI_Interface_Overview".homeCodition[13].emOverviewCmName[9] := WSTRING#'Spare';
           "HMI_Interface_Overview".homeCodition[13].emOverviewCmName[10] := WSTRING#'Spare';
           "HMI_Interface_Overview".homeCodition[13].emOverviewCmName[11] := WSTRING#'Spare';
           "HMI_Interface_Overview".homeCodition[13].emOverviewCmName[12] := WSTRING#'Spare';
           "HMI_Interface_Overview".homeCodition[13].emOverviewCmName[13] := WSTRING#'Spare';
           "HMI_Interface_Overview".homeCodition[13].emOverviewCmPositionName[0] := WSTRING#'Wait Position';
           "HMI_Interface_Overview".homeCodition[13].emOverviewCmPositionName[1] := WSTRING#'Wait Position';
           "HMI_Interface_Overview".homeCodition[13].emOverviewCmPositionName[2] := WSTRING#'Wait Position';
           "HMI_Interface_Overview".homeCodition[13].emOverviewCmPositionName[3] := WSTRING#'Open';
           "HMI_Interface_Overview".homeCodition[13].emOverviewCmPositionName[4] := WSTRING#'Not Detect';
           "HMI_Interface_Overview".homeCodition[13].emOverviewCmPositionName[5] := WSTRING#'Spare';
           "HMI_Interface_Overview".homeCodition[13].emOverviewCmPositionName[6] := WSTRING#'Spare';
           "HMI_Interface_Overview".homeCodition[13].emOverviewCmPositionName[7] := WSTRING#'Spare';
           "HMI_Interface_Overview".homeCodition[13].emOverviewCmPositionName[8] := WSTRING#'Spare';
           "HMI_Interface_Overview".homeCodition[13].emOverviewCmPositionName[9] := WSTRING#'Spare';
           "HMI_Interface_Overview".homeCodition[13].emOverviewCmPositionName[10] := WSTRING#'Spare';
           "HMI_Interface_Overview".homeCodition[13].emOverviewCmPositionName[11] := WSTRING#'Spare';
           "HMI_Interface_Overview".homeCodition[13].emOverviewCmPositionName[12] := WSTRING#'Spare';
           "HMI_Interface_Overview".homeCodition[13].emOverviewCmPositionName[13] := WSTRING#'Spare';
           IF NOT #statLampControl THEN
               "HMI_Interface_Overview".homeCodition[13].emOverviewHomeLampOn[0] := "Unit1.Em13.HmiInterface".cm.softcam.jrUnIoadingPnPAxisX.pos00_wait.inPos;
               "HMI_Interface_Overview".homeCodition[13].emOverviewHomeLampOn[1] := "Unit1.Em13.HmiInterface".cm.softcam.jrUnIoadingPnPAxisZ.pos00_wait.inPos;
               "HMI_Interface_Overview".homeCodition[13].emOverviewHomeLampOn[2] := "Unit1.Em13.HmiInterface".cm.softcam.jrUnIoadingPnPAxisC.pos00_wait.inPos;
               "HMI_Interface_Overview".homeCodition[13].emOverviewHomeLampOn[3] := "Unit1.Em13.HmiInterface".cmJRUnloadingPnPClampOpenClose.monitoring.inHomePos;
               "HMI_Interface_Overview".homeCodition[13].emOverviewHomeLampOn[4] := NOT "Unit1.Em13.HmiInterface".cmJRUnloadingPnPJRDetect.monitoring.processValue;
               "HMI_Interface_Overview".homeCodition[13].emOverviewHomeLampOn[5] := FALSE;
               "HMI_Interface_Overview".homeCodition[13].emOverviewHomeLampOn[6] := FALSE;
               "HMI_Interface_Overview".homeCodition[13].emOverviewHomeLampOn[7] := FALSE;
               "HMI_Interface_Overview".homeCodition[13].emOverviewHomeLampOn[8] := FALSE;
               "HMI_Interface_Overview".homeCodition[13].emOverviewHomeLampOn[9] := FALSE;
               "HMI_Interface_Overview".homeCodition[13].emOverviewHomeLampOn[10] := FALSE;
               "HMI_Interface_Overview".homeCodition[13].emOverviewHomeLampOn[11] := FALSE;
               "HMI_Interface_Overview".homeCodition[13].emOverviewHomeLampOn[12] := FALSE;
               "HMI_Interface_Overview".homeCodition[13].emOverviewHomeLampOn[13] := FALSE;
           END_IF;
       END_IF;

       // Index 1
       IF "HMI_Interface_Overview".homeCodition[13].pageIndex = 1 THEN
           "HMI_Interface_Overview".homeCodition[13].emOverviewTitle := WSTRING#'Home Condition 1';
           "HMI_Interface_Overview".homeCodition[13].emOverviewCmName[0] := WSTRING#'JR Unloading P&P X-Axis';
           "HMI_Interface_Overview".homeCodition[13].emOverviewCmName[1] := WSTRING#'JR Unloading P&P Z-Axis';
           "HMI_Interface_Overview".homeCodition[13].emOverviewCmName[2] := WSTRING#'JR Unloading P&P C-Axis';
           "HMI_Interface_Overview".homeCodition[13].emOverviewCmName[3] := WSTRING#'JR Unloading P&P Clamp';
           "HMI_Interface_Overview".homeCodition[13].emOverviewCmName[4] := WSTRING#'JR Unloading P&P JR Detect';
           "HMI_Interface_Overview".homeCodition[13].emOverviewCmName[5] := WSTRING#'Spare';
           "HMI_Interface_Overview".homeCodition[13].emOverviewCmName[6] := WSTRING#'Spare';
           "HMI_Interface_Overview".homeCodition[13].emOverviewCmName[7] := WSTRING#'Spare';
           "HMI_Interface_Overview".homeCodition[13].emOverviewCmName[8] := WSTRING#'Spare';
           "HMI_Interface_Overview".homeCodition[13].emOverviewCmName[9] := WSTRING#'Spare';
           "HMI_Interface_Overview".homeCodition[13].emOverviewCmName[10] := WSTRING#'Spare';
           "HMI_Interface_Overview".homeCodition[13].emOverviewCmName[11] := WSTRING#'Spare';
           "HMI_Interface_Overview".homeCodition[13].emOverviewCmName[12] := WSTRING#'Spare';
           "HMI_Interface_Overview".homeCodition[13].emOverviewCmName[13] := WSTRING#'Spare';
           "HMI_Interface_Overview".homeCodition[13].emOverviewCmPositionName[0] := WSTRING#'Wait Position';
           "HMI_Interface_Overview".homeCodition[13].emOverviewCmPositionName[1] := WSTRING#'Wait Position';
           "HMI_Interface_Overview".homeCodition[13].emOverviewCmPositionName[2] := WSTRING#'Wait Position';
           "HMI_Interface_Overview".homeCodition[13].emOverviewCmPositionName[3] := WSTRING#'Close';
           "HMI_Interface_Overview".homeCodition[13].emOverviewCmPositionName[4] := WSTRING#'Detect';
           "HMI_Interface_Overview".homeCodition[13].emOverviewCmPositionName[5] := WSTRING#'Spare';
           "HMI_Interface_Overview".homeCodition[13].emOverviewCmPositionName[6] := WSTRING#'Spare';
           "HMI_Interface_Overview".homeCodition[13].emOverviewCmPositionName[7] := WSTRING#'Spare';
           "HMI_Interface_Overview".homeCodition[13].emOverviewCmPositionName[8] := WSTRING#'Spare';
           "HMI_Interface_Overview".homeCodition[13].emOverviewCmPositionName[9] := WSTRING#'Spare';
           "HMI_Interface_Overview".homeCodition[13].emOverviewCmPositionName[10] := WSTRING#'Spare';
           "HMI_Interface_Overview".homeCodition[13].emOverviewCmPositionName[11] := WSTRING#'Spare';
           "HMI_Interface_Overview".homeCodition[13].emOverviewCmPositionName[12] := WSTRING#'Spare';
           "HMI_Interface_Overview".homeCodition[13].emOverviewCmPositionName[13] := WSTRING#'Spare';
           IF NOT #statLampControl THEN
               "HMI_Interface_Overview".homeCodition[13].emOverviewHomeLampOn[0] := "Unit1.Em13.HmiInterface".cm.softcam.jrUnIoadingPnPAxisX.pos00_wait.inPos;
               "HMI_Interface_Overview".homeCodition[13].emOverviewHomeLampOn[1] := "Unit1.Em13.HmiInterface".cm.softcam.jrUnIoadingPnPAxisZ.pos00_wait.inPos;
               "HMI_Interface_Overview".homeCodition[13].emOverviewHomeLampOn[2] := "Unit1.Em13.HmiInterface".cm.softcam.jrUnIoadingPnPAxisC.pos00_wait.inPos;
               "HMI_Interface_Overview".homeCodition[13].emOverviewHomeLampOn[3] := "Unit1.Em13.HmiInterface".cmJRUnloadingPnPClampOpenClose.monitoring.inWorkPos;
               "HMI_Interface_Overview".homeCodition[13].emOverviewHomeLampOn[4] := "Unit1.Em13.HmiInterface".cmJRUnloadingPnPJRDetect.monitoring.processValue;
               "HMI_Interface_Overview".homeCodition[13].emOverviewHomeLampOn[5] := FALSE;
               "HMI_Interface_Overview".homeCodition[13].emOverviewHomeLampOn[6] := FALSE;
               "HMI_Interface_Overview".homeCodition[13].emOverviewHomeLampOn[7] := FALSE;
               "HMI_Interface_Overview".homeCodition[13].emOverviewHomeLampOn[8] := FALSE;
               "HMI_Interface_Overview".homeCodition[13].emOverviewHomeLampOn[9] := FALSE;
               "HMI_Interface_Overview".homeCodition[13].emOverviewHomeLampOn[10] := FALSE;
               "HMI_Interface_Overview".homeCodition[13].emOverviewHomeLampOn[11] := FALSE;
               "HMI_Interface_Overview".homeCodition[13].emOverviewHomeLampOn[12] := FALSE;
               "HMI_Interface_Overview".homeCodition[13].emOverviewHomeLampOn[13] := FALSE;
           END_IF;
       END_IF;

   END_REGION
END_REGION
END_FUNCTION_BLOCK

FUNCTION "ParameterMove" : Void   // FC26, LAD
// stored: SetENOAutomatically false
   VAR_TEMP
      tempSoftCamIndex : Int;
   END_VAR
   VAR_TEMP   // added for the SCL form of the ladder/FBD networks
      _w1 : Bool;
      _w2 : Bool;
      _w3 : Bool;
      _w4 : Bool;
      _w5 : Bool;
      _w6 : Bool;
      _w7 : Bool;
      _w8 : Bool;
      _w9 : Bool;
      _w10 : Bool;
      _w11 : Bool;
      _w12 : Bool;
      _w13 : Bool;
      _w14 : Bool;
   END_VAR
BEGIN

REGION Network 1 (SCL): Recipe → HMI | Read |
END_REGION

REGION Network 2 (SCL): HMI → PLC | Apply | Softcam_unuse_0420
   //IF "HMI_Interface_Parameter".RecipeButton.Apply THEN
   //    FOR #tempSoftCamIndex := 0 TO 15 DO
   //        Unit1.Em2.HmiInterface.cm.softcam.jrOutPnPLeftAxisX.position[#tempSoftCamIndex].SetValue := "HMI_Interface_Parameter".Softcam[1].position[#tempSoftCamIndex].SetValue;
   //        Unit1.Em2.HmiInterface.cm.softcam.jrOutPnPLeftAxisZ.position[#tempSoftCamIndex].SetValue := "HMI_Interface_Parameter".Softcam[2].position[#tempSoftCamIndex].SetValue;
   //        Unit1.Em2.HmiInterface.cm.softcam.jrOutPnPRightAxisX.position[#tempSoftCamIndex].SetValue := "HMI_Interface_Parameter".Softcam[3].position[#tempSoftCamIndex].SetValue;
   //        Unit1.Em2.HmiInterface.cm.softcam.jrOutPnPRightAxisZ.position[#tempSoftCamIndex].SetValue := "HMI_Interface_Parameter".Softcam[4].position[#tempSoftCamIndex].SetValue;

           //        Unit1.Em3.HmiInterface.cm.softcam.topTapeAxisX.position[#tempSoftCamIndex].SetValue := "HMI_Interface_Parameter".Softcam[5].position[#tempSoftCamIndex].SetValue;
           //        Unit1.Em3.HmiInterface.cm.softcam.topTapeAxisY.position[#tempSoftCamIndex].SetValue := "HMI_Interface_Parameter".Softcam[6].position[#tempSoftCamIndex].SetValue;

           //        Unit1.Em4.HmiInterface.cm.softcam.sideTapeFixStageAxisX.position[#tempSoftCamIndex].SetValue := "HMI_Interface_Parameter".Softcam[7].position[#tempSoftCamIndex].SetValue;
           //        Unit1.Em4.HmiInterface.cm.softcam.sideTapeFixStageAxisC.position[#tempSoftCamIndex].SetValue := "HMI_Interface_Parameter".Softcam[8].position[#tempSoftCamIndex].SetValue;
           //        Unit1.Em4.HmiInterface.cm.softcam.sideTapeAttachmentAxisX.position[#tempSoftCamIndex].SetValue := "HMI_Interface_Parameter".Softcam[9].position[#tempSoftCamIndex].SetValue;
           //        Unit1.Em4.HmiInterface.cm.softcam.sideTapeAttachmentAxisY.position[#tempSoftCamIndex].SetValue := "HMI_Interface_Parameter".Softcam[10].position[#tempSoftCamIndex].SetValue;

           //        Unit1.Em5.HmiInterface.cm.softcam.transferPnPLeftAxisX.position[#tempSoftCamIndex].SetValue := "HMI_Interface_Parameter".Softcam[11].position[#tempSoftCamIndex].SetValue;
           //        Unit1.Em5.HmiInterface.cm.softcam.transferPnPLeftAxisY.position[#tempSoftCamIndex].SetValue := "HMI_Interface_Parameter".Softcam[12].position[#tempSoftCamIndex].SetValue;
           //        Unit1.Em5.HmiInterface.cm.softcam.transferPnPLeftAxisZ.position[#tempSoftCamIndex].SetValue := "HMI_Interface_Parameter".Softcam[13].position[#tempSoftCamIndex].SetValue;
           //        Unit1.Em5.HmiInterface.cm.softcam.transferPnPRightAxisX.position[#tempSoftCamIndex].SetValue := "HMI_Interface_Parameter".Softcam[14].position[#tempSoftCamIndex].SetValue;
           //        Unit1.Em5.HmiInterface.cm.softcam.transferPnPRightAxisY.position[#tempSoftCamIndex].SetValue := "HMI_Interface_Parameter".Softcam[15].position[#tempSoftCamIndex].SetValue;
           //        Unit1.Em5.HmiInterface.cm.softcam.transferPnPRightAxisZ.position[#tempSoftCamIndex].SetValue := "HMI_Interface_Parameter".Softcam[16].position[#tempSoftCamIndex].SetValue;

           //        Unit1.Em8.HmiInterface.cm.softcam.thicknessAxisZ.position[#tempSoftCamIndex].SetValue := "HMI_Interface_Parameter".Softcam[17].position[#tempSoftCamIndex].SetValue;

           //        Unit1.Em13.HmiInterface.cm.softcam.jrUnloadingPnPAxisX.position[#tempSoftCamIndex].SetValue := "HMI_Interface_Parameter".Softcam[18].position[#tempSoftCamIndex].SetValue;
           //        Unit1.Em13.HmiInterface.cm.softcam.jrUnloadingPnPAxisZ.position[#tempSoftCamIndex].SetValue := "HMI_Interface_Parameter".Softcam[19].position[#tempSoftCamIndex].SetValue;
           //        Unit1.Em13.HmiInterface.cm.softcam.jrUnloadingPnPAxisC.position[#tempSoftCamIndex].SetValue := "HMI_Interface_Parameter".Softcam[20].position[#tempSoftCamIndex].SetValue;
           //    END_FOR;
           //END_IF;
END_REGION

REGION Network 3 (SCL): HMI → PLC | Apply | Parameter
   IF "HMI_Interface_Parameter".RecipeButton.Apply THEN

       "HMI_Interface_Parameter".Parameter[0]."Process Value" := "HMI_Interface_Parameter".Parameter[0]."Set Value"; // Sleep Mode Activation Time
       "Unit1.EmNodes".SleepModeActivationTime := DINT_TO_TIME(ROUND("HMI_Interface_Parameter".Parameter[0]."Process Value" * 60000.0));

       "HMI_Interface_Parameter".Parameter[1]."Process Value" := "HMI_Interface_Parameter".Parameter[1]."Set Value"; // Deep Sleep Mode Activation Time
       "Unit1.EmNodes".DeepSleepModeActivationTime := DINT_TO_TIME(ROUND("HMI_Interface_Parameter".Parameter[1]."Process Value" * 60000.0));

       "HMI_Interface_Parameter".Parameter[2]."Process Value" := "HMI_Interface_Parameter".Parameter[2]."Set Value"; // FFU_sleepmoderunpct
       "Unit1.HmiInterface".FFU_SleepModeRunPct := LREAL_TO_INT("HMI_Interface_Parameter".Parameter[2]."Set Value");

   END_IF;

   "Unit1.Em2.HmiInterface".cm.distance.setValue.distanceLimitSV := "RecipeParameter".ParameterPV.Recipe1; // BA060AZSIDR1_JROutP&PLeftAxisX ↔ BA060AZSIDR3_JROutP&PRightAxisX
   "Unit1.Em5.HmiInterface".cm.distance.setValue.distanceLimitSV := "RecipeParameter".ParameterPV.Recipe2; // BA060AZSIDR12_TransferP&PLeftAxisX ↔ BA060AZSIDR15_TransferP&PRightAxisX
   "Unit1.Em9.HmiInterface".gaugeRnR.processCount := LREAL_TO_INT(IN := "RecipeParameter".ParameterPV."Recipe3"); // Vision R&R
   "Unit1.Em8.HmiInterface".gaugeRnR.processCount := LREAL_TO_INT(IN := "RecipeParameter".ParameterPV.Recipe4); // Thickness R&R
   "Unit1.Em8.HmiInterface".HipotRepeat.processCount := LREAL_TO_INT(IN := "RecipeParameter".ParameterPV."Recipe5"); // Hipot Repeat SV
   "Unit1.Em3.HmiInterface".TopTapeIdleTime.processCount := DINT_TO_TIME(ROUND(IN := "RecipeParameter".ParameterPV."Recipe6")); // TopTape IDLE Time
   "Unit1.Em4.HmiInterface".SideTapeIdleTime.processCount := DINT_TO_TIME(ROUND(IN := "RecipeParameter".ParameterPV."Recipe7")); // SideTape IDLE Time
   "Unit1.Em9.HmiInterface".VisionRetryCount.processCount := LREAL_TO_INT(IN := "RecipeParameter".ParameterPV."Recipe8"); // Vision NG Retry Count
END_REGION

REGION Network 4 (SCL): HMI → PLC | Apply | FAT Mode
   IF "HMI_Interface_Parameter".RecipeButton.Apply THEN
       "Unit1.EmNodes".FATModeInterface.HoursTest.ProcessValue.SelectHours_ProcessValue := "HMI_Interface_Parameter".FATModeInterface.HoursTest.ProcessValue.SelectHours_ProcessValue := "HMI_Interface_Parameter".FATModeInterface.HoursTest.SetValue.SelectHours_SetValue;
       "Unit1.EmNodes".FATModeInterface.Capability.ProcessValue.SelectCycle_ProcessValue := "HMI_Interface_Parameter".FATModeInterface.Capability.ProcessValue.SelectCycle_ProcessValue := "HMI_Interface_Parameter".FATModeInterface.Capability.SetValue.SelectCycle_SetValue;
       "Unit1.EmNodes".FATModeInterface.Sampling.ProcessValue.SelectCount_ProcessValue := "HMI_Interface_Parameter".FATModeInterface.Sampling.ProcessValue.SelectCount_ProcessValue := "HMI_Interface_Parameter".FATModeInterface.Sampling.SetValue.SelectCount_SetValue;
   END_IF;
END_REGION

REGION Network 5 (SCL): HMI → PLC | Button | FAT Mode
   // FAT Parameter
   "Unit1.EmNodes".FATModeSelect.HoursTestMode := "HMI_Interface_Parameter".FATModeSelect.HoursTestMode;
   "Unit1.EmNodes".FATModeSelect.CapabilityMode := "HMI_Interface_Parameter".FATModeSelect.CapabilityMode;
   "Unit1.EmNodes".FATModeSelect.SamplingMode := "HMI_Interface_Parameter".FATModeSelect.SamplingMode;

   // FAT Mode Sampling Clear And Select Interlock
   IF "Unit1.EmNodes".FATModeSelect.SamplingMode AND "Unit1.EmNodes".SamplingModeComplete THEN
       "HMI_Interface_Parameter".FATModeSelect.SamplingMode := FALSE;
   // ELSIF Unit1.EmNodes.unitStatus.specialFunctions.dryRun THEN
   //     "HMI_Interface_Parameter".FATModeSelect.SamplingMode := FALSE;
   //     "HMI_Interface_Parameter".FATModeSelect.CapabilityMode := FALSE;
   END_IF;
END_REGION

REGION Network 6 (SCL): PLC → HMI | Always | Softcam_unuse_0420
   //FOR #tempSoftCamIndex := 0 TO 15 DO
   //    "HMI_Interface_Parameter".Softcam[1].TargetPosition := Unit1.Em2.HmiInterface.cm.softcam.jrOutPnPLeftAxisX.TargetPosition;
   //    "HMI_Interface_Parameter".Softcam[1].ActualPosition := Unit1.Em2.HmiInterface.cm.softcam.jrOutPnPLeftAxisX.ActualPosition;
   //    "HMI_Interface_Parameter".Softcam[2].TargetPosition := Unit1.Em2.HmiInterface.cm.softcam.jrOutPnPLeftAxisZ.TargetPosition;
   //    "HMI_Interface_Parameter".Softcam[2].ActualPosition := Unit1.Em2.HmiInterface.cm.softcam.jrOutPnPLeftAxisZ.ActualPosition;
   //    "HMI_Interface_Parameter".Softcam[3].TargetPosition := Unit1.Em2.HmiInterface.cm.softcam.jrOutPnPRightAxisX.TargetPosition;
   //    "HMI_Interface_Parameter".Softcam[3].ActualPosition := Unit1.Em2.HmiInterface.cm.softcam.jrOutPnPRightAxisX.ActualPosition;
   //    "HMI_Interface_Parameter".Softcam[4].TargetPosition := Unit1.Em2.HmiInterface.cm.softcam.jrOutPnPRightAxisZ.TargetPosition;
   //    "HMI_Interface_Parameter".Softcam[4].ActualPosition := Unit1.Em2.HmiInterface.cm.softcam.jrOutPnPRightAxisZ.ActualPosition;

   //    "HMI_Interface_Parameter".Softcam[5].TargetPosition := Unit1.Em3.HmiInterface.cm.softcam.topTapeAxisX.TargetPosition;
   //    "HMI_Interface_Parameter".Softcam[5].ActualPosition := Unit1.Em3.HmiInterface.cm.softcam.topTapeAxisX.ActualPosition;
   //    "HMI_Interface_Parameter".Softcam[6].TargetPosition := Unit1.Em3.HmiInterface.cm.softcam.topTapeAxisY.TargetPosition;
   //    "HMI_Interface_Parameter".Softcam[6].ActualPosition := Unit1.Em3.HmiInterface.cm.softcam.topTapeAxisY.ActualPosition;

   //   "HMI_Interface_Parameter".Softcam[7].TargetPosition := Unit1.Em4.HmiInterface.cm.softcam.sideTapeFixStageAxisX.TargetPosition;
   //    "HMI_Interface_Parameter".Softcam[7].ActualPosition := Unit1.Em4.HmiInterface.cm.softcam.sideTapeFixStageAxisX.ActualPosition;
   //    "HMI_Interface_Parameter".Softcam[8].TargetPosition := Unit1.Em4.HmiInterface.cm.softcam.sideTapeFixStageAxisC.TargetPosition;
   //    "HMI_Interface_Parameter".Softcam[8].ActualPosition := Unit1.Em4.HmiInterface.cm.softcam.sideTapeFixStageAxisC.ActualPosition;
   //    "HMI_Interface_Parameter".Softcam[9].TargetPosition := Unit1.Em4.HmiInterface.cm.softcam.sideTapeAttachmentAxisX.TargetPosition;
   //    "HMI_Interface_Parameter".Softcam[9].ActualPosition := Unit1.Em4.HmiInterface.cm.softcam.sideTapeAttachmentAxisX.ActualPosition;
   //    "HMI_Interface_Parameter".Softcam[10].TargetPosition := Unit1.Em4.HmiInterface.cm.softcam.sideTapeAttachmentAxisY.TargetPosition;
   //    "HMI_Interface_Parameter".Softcam[10].ActualPosition := Unit1.Em4.HmiInterface.cm.softcam.sideTapeAttachmentAxisY.ActualPosition;

   //    "HMI_Interface_Parameter".Softcam[11].TargetPosition := Unit1.Em5.HmiInterface.cm.softcam.transferPnPLeftAxisX.TargetPosition;
   //    "HMI_Interface_Parameter".Softcam[11].ActualPosition := Unit1.Em5.HmiInterface.cm.softcam.transferPnPLeftAxisX.ActualPosition;
   //    "HMI_Interface_Parameter".Softcam[12].TargetPosition := Unit1.Em5.HmiInterface.cm.softcam.transferPnPLeftAxisY.TargetPosition;
   //    "HMI_Interface_Parameter".Softcam[12].ActualPosition := Unit1.Em5.HmiInterface.cm.softcam.transferPnPLeftAxisY.ActualPosition;
   //    "HMI_Interface_Parameter".Softcam[13].TargetPosition := Unit1.Em5.HmiInterface.cm.softcam.transferPnPLeftAxisZ.TargetPosition;
   //    "HMI_Interface_Parameter".Softcam[13].ActualPosition := Unit1.Em5.HmiInterface.cm.softcam.transferPnPLeftAxisZ.ActualPosition;
   //    "HMI_Interface_Parameter".Softcam[14].TargetPosition := Unit1.Em5.HmiInterface.cm.softcam.transferPnPRightAxisX.TargetPosition;
   //    "HMI_Interface_Parameter".Softcam[14].ActualPosition := Unit1.Em5.HmiInterface.cm.softcam.transferPnPRightAxisX.ActualPosition;
   //    "HMI_Interface_Parameter".Softcam[15].TargetPosition := Unit1.Em5.HmiInterface.cm.softcam.transferPnPRightAxisY.TargetPosition;
   //    "HMI_Interface_Parameter".Softcam[15].ActualPosition := Unit1.Em5.HmiInterface.cm.softcam.transferPnPRightAxisY.ActualPosition;
   //    "HMI_Interface_Parameter".Softcam[16].TargetPosition := Unit1.Em5.HmiInterface.cm.softcam.transferPnPRightAxisZ.TargetPosition;
   //    "HMI_Interface_Parameter".Softcam[16].ActualPosition := Unit1.Em5.HmiInterface.cm.softcam.transferPnPRightAxisZ.ActualPosition;

   //    "HMI_Interface_Parameter".Softcam[17].TargetPosition := Unit1.Em8.HmiInterface.cm.softcam.thicknessAxisZ.TargetPosition;
   //    "HMI_Interface_Parameter".Softcam[17].ActualPosition := Unit1.Em8.HmiInterface.cm.softcam.thicknessAxisZ.ActualPosition;

   //    "HMI_Interface_Parameter".Softcam[18].TargetPosition := Unit1.Em13.HmiInterface.cm.softcam.jrUnloadingPnPAxisX.TargetPosition;
   //    "HMI_Interface_Parameter".Softcam[18].ActualPosition := Unit1.Em13.HmiInterface.cm.softcam.jrUnloadingPnPAxisX.ActualPosition;
   //    "HMI_Interface_Parameter".Softcam[19].TargetPosition := Unit1.Em13.HmiInterface.cm.softcam.jrUnloadingPnPAxisZ.TargetPosition;
   //    "HMI_Interface_Parameter".Softcam[19].ActualPosition := Unit1.Em13.HmiInterface.cm.softcam.jrUnloadingPnPAxisZ.ActualPosition;
   //    "HMI_Interface_Parameter".Softcam[20].TargetPosition := Unit1.Em13.HmiInterface.cm.softcam.jrUnloadingPnPAxisC.TargetPosition;
   //    "HMI_Interface_Parameter".Softcam[20].ActualPosition := Unit1.Em13.HmiInterface.cm.softcam.jrUnloadingPnPAxisC.ActualPosition;

   //    "HMI_Interface_Parameter".Softcam[1].position[#tempSoftCamIndex].ProcessValue := Unit1.Em2.HmiInterface.cm.softcam.jrOutPnPLeftAxisX.position[#tempSoftCamIndex].ProcessValue;
   //    "HMI_Interface_Parameter".Softcam[2].position[#tempSoftCamIndex].ProcessValue := Unit1.Em2.HmiInterface.cm.softcam.jrOutPnPLeftAxisZ.position[#tempSoftCamIndex].ProcessValue;
   //    "HMI_Interface_Parameter".Softcam[3].position[#tempSoftCamIndex].ProcessValue := Unit1.Em2.HmiInterface.cm.softcam.jrOutPnPRightAxisX.position[#tempSoftCamIndex].ProcessValue;
   //    "HMI_Interface_Parameter".Softcam[4].position[#tempSoftCamIndex].ProcessValue := Unit1.Em2.HmiInterface.cm.softcam.jrOutPnPRightAxisZ.position[#tempSoftCamIndex].ProcessValue;

   //    "HMI_Interface_Parameter".Softcam[5].position[#tempSoftCamIndex].ProcessValue := Unit1.Em3.HmiInterface.cm.softcam.topTapeAxisX.position[#tempSoftCamIndex].ProcessValue;
   //    "HMI_Interface_Parameter".Softcam[6].position[#tempSoftCamIndex].ProcessValue := Unit1.Em3.HmiInterface.cm.softcam.topTapeAxisY.position[#tempSoftCamIndex].ProcessValue;

   //    "HMI_Interface_Parameter".Softcam[7].position[#tempSoftCamIndex].ProcessValue := Unit1.Em4.HmiInterface.cm.softcam.sideTapeFixStageAxisX.position[#tempSoftCamIndex].ProcessValue;
   //    "HMI_Interface_Parameter".Softcam[8].position[#tempSoftCamIndex].ProcessValue := Unit1.Em4.HmiInterface.cm.softcam.sideTapeFixStageAxisC.position[#tempSoftCamIndex].ProcessValue;
   //    "HMI_Interface_Parameter".Softcam[9].position[#tempSoftCamIndex].ProcessValue := Unit1.Em4.HmiInterface.cm.softcam.sideTapeAttachmentAxisX.position[#tempSoftCamIndex].ProcessValue;
   //    "HMI_Interface_Parameter".Softcam[10].position[#tempSoftCamIndex].ProcessValue := Unit1.Em4.HmiInterface.cm.softcam.sideTapeAttachmentAxisY.position[#tempSoftCamIndex].ProcessValue;

   //    "HMI_Interface_Parameter".Softcam[11].position[#tempSoftCamIndex].ProcessValue := Unit1.Em5.HmiInterface.cm.softcam.transferPnPLeftAxisX.position[#tempSoftCamIndex].ProcessValue;
   //    "HMI_Interface_Parameter".Softcam[12].position[#tempSoftCamIndex].ProcessValue := Unit1.Em5.HmiInterface.cm.softcam.transferPnPLeftAxisY.position[#tempSoftCamIndex].ProcessValue;
   //    "HMI_Interface_Parameter".Softcam[13].position[#tempSoftCamIndex].ProcessValue := Unit1.Em5.HmiInterface.cm.softcam.transferPnPLeftAxisZ.position[#tempSoftCamIndex].ProcessValue;
   //    "HMI_Interface_Parameter".Softcam[14].position[#tempSoftCamIndex].ProcessValue := Unit1.Em5.HmiInterface.cm.softcam.transferPnPRightAxisX.position[#tempSoftCamIndex].ProcessValue;
   //    "HMI_Interface_Parameter".Softcam[15].position[#tempSoftCamIndex].ProcessValue := Unit1.Em5.HmiInterface.cm.softcam.transferPnPRightAxisY.position[#tempSoftCamIndex].ProcessValue;
   //    "HMI_Interface_Parameter".Softcam[16].position[#tempSoftCamIndex].ProcessValue := Unit1.Em5.HmiInterface.cm.softcam.transferPnPRightAxisZ.position[#tempSoftCamIndex].ProcessValue;

   //    "HMI_Interface_Parameter".Softcam[17].position[#tempSoftCamIndex].ProcessValue := Unit1.Em8.HmiInterface.cm.softcam.thicknessAxisZ.position[#tempSoftCamIndex].ProcessValue;

   //    "HMI_Interface_Parameter".Softcam[18].position[#tempSoftCamIndex].ProcessValue := Unit1.Em13.HmiInterface.cm.softcam.jrUnloadingPnPAxisX.position[#tempSoftCamIndex].ProcessValue;
   //    "HMI_Interface_Parameter".Softcam[19].position[#tempSoftCamIndex].ProcessValue := Unit1.Em13.HmiInterface.cm.softcam.jrUnloadingPnPAxisZ.position[#tempSoftCamIndex].ProcessValue;
   //    "HMI_Interface_Parameter".Softcam[20].position[#tempSoftCamIndex].ProcessValue := Unit1.Em13.HmiInterface.cm.softcam.jrUnloadingPnPAxisC.position[#tempSoftCamIndex].ProcessValue;
   //END_FOR;
   //

   "HMI_Interface_Parameter".Softcam[1] := "Unit1.Em2.HmiInterface".cm.softcam.jrOutPnPLeftAxisX;
   "HMI_Interface_Parameter".Softcam[2] := "Unit1.Em2.HmiInterface".cm.softcam.jrOutPnPLeftAxisZ;
   "HMI_Interface_Parameter".Softcam[3] := "Unit1.Em2.HmiInterface".cm.softcam.jrOutPnPRightAxisX;
   "HMI_Interface_Parameter".Softcam[4] := "Unit1.Em2.HmiInterface".cm.softcam.jrOutPnPRightAxisZ;
   "HMI_Interface_Parameter".Softcam[5] := "Unit1.Em3.HmiInterface".cm.softcam.topTapeAxisX;
   "HMI_Interface_Parameter".Softcam[6] := "Unit1.Em3.HmiInterface".cm.softcam.topTapeAxisY;
   "HMI_Interface_Parameter".Softcam[7] := "Unit1.Em4.HmiInterface".cm.softcam.sideTapeFixStageAxisX;
   "HMI_Interface_Parameter".Softcam[8] := "Unit1.Em4.HmiInterface".cm.softcam.sideTapeFixStageAxisC;
   "HMI_Interface_Parameter".Softcam[9] := "Unit1.Em4.HmiInterface".cm.softcam.sideTapeAttachmentAxisX;
   "HMI_Interface_Parameter".Softcam[10] := "Unit1.Em4.HmiInterface".cm.softcam.sideTapeAttachmentAxisY;
   "HMI_Interface_Parameter".Softcam[11] := "Unit1.Em5.HmiInterface".cm.softcam.transferPnPLeftAxisX;
   "HMI_Interface_Parameter".Softcam[12] := "Unit1.Em5.HmiInterface".cm.softcam.transferPnPLeftAxisY;
   "HMI_Interface_Parameter".Softcam[13] := "Unit1.Em5.HmiInterface".cm.softcam.transferPnPLeftAxisZ;
   "HMI_Interface_Parameter".Softcam[14] := "Unit1.Em5.HmiInterface".cm.softcam.transferPnPRightAxisX;
   "HMI_Interface_Parameter".Softcam[15] := "Unit1.Em5.HmiInterface".cm.softcam.transferPnPRightAxisY;
   "HMI_Interface_Parameter".Softcam[16] := "Unit1.Em5.HmiInterface".cm.softcam.transferPnPRightAxisZ;
   "HMI_Interface_Parameter".Softcam[17] := "Unit1.Em8.HmiInterface".cm.softcam.thicknessAxisZ;
   "HMI_Interface_Parameter".Softcam[18] := "Unit1.Em13.HmiInterface".cm.softcam.jrUnIoadingPnPAxisX;
   "HMI_Interface_Parameter".Softcam[19] := "Unit1.Em13.HmiInterface".cm.softcam.jrUnIoadingPnPAxisZ;
   "HMI_Interface_Parameter".Softcam[20] := "Unit1.Em13.HmiInterface".cm.softcam.jrUnIoadingPnPAxisC;
END_REGION

REGION Network 7 (SCL): PLC → HMI | Always | Distance
   // "RecipeParameter".ParameterPV."Recipe1" := Unit1.Em2.HmiInterface.cm.distance.processValue.distanceLimitPV; // BA060AZSIDR1_JROutP&PLeftAxisX ↔ BA060AZSIDR3_JROutP&PRightAxisX
   // "RecipeParameter".ParameterPV."Recipe2" := Unit1.Em5.HmiInterface.cm.distance.processValue.distanceLimitPV; // BA060AZSIDR12_TransferP&PLeftAxisX ↔ BA060AZSIDR15_TransferP&PRightAxisX
END_REGION

REGION Network 8 (SCL): PLC → HMI | Always | FAT Mode
   // FAT Parameter
   "HMI_Interface_Parameter".FATModeInterface.HoursTest.ProcessValue.ProcTimeLeft := "Unit1.EmNodes".FATModeInterface.HoursTest.ProcessValue.ProcTimeLeft;
   "HMI_Interface_Parameter".FATModeInterface.Capability.ProcessValue.CapabilityCount := "Unit1.EmNodes".FATModeInterface.Capability.ProcessValue.CapabilityCount;
   "HMI_Interface_Parameter".FATModeInterface.Sampling.ProcessValue.CellCount := "Unit1.EmNodes".FATModeInterface.Sampling.ProcessValue.CellCount;
END_REGION

REGION Network 9: Call Recipe
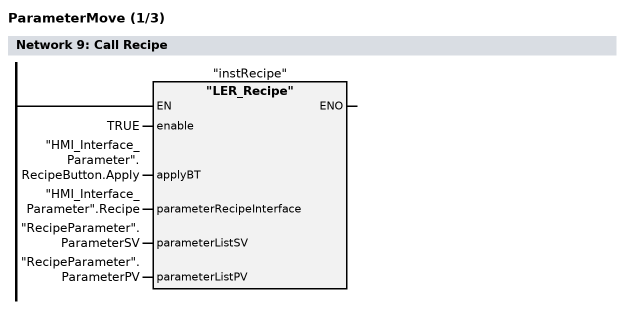
   RUNG wire#powerrail
      "instRecipe"(enable := TRUE, applyBT := "HMI_Interface_Parameter".RecipeButton.Apply, parameterRecipeInterface := "HMI_Interface_Parameter".Recipe, parameterListSV := "RecipeParameter".ParameterSV, parameterListPV := "RecipeParameter".ParameterPV)
   END_RUNG
   // the same network as SCL:
   "instRecipe"(enable := TRUE,   // "LER_Recipe"
                applyBT := "HMI_Interface_Parameter".RecipeButton.Apply,
                parameterRecipeInterface := "HMI_Interface_Parameter".Recipe,
                parameterListSV := "RecipeParameter".ParameterSV,
                parameterListPV := "RecipeParameter".ParameterPV);
END_REGION

REGION Network 10: Call Teaching Position
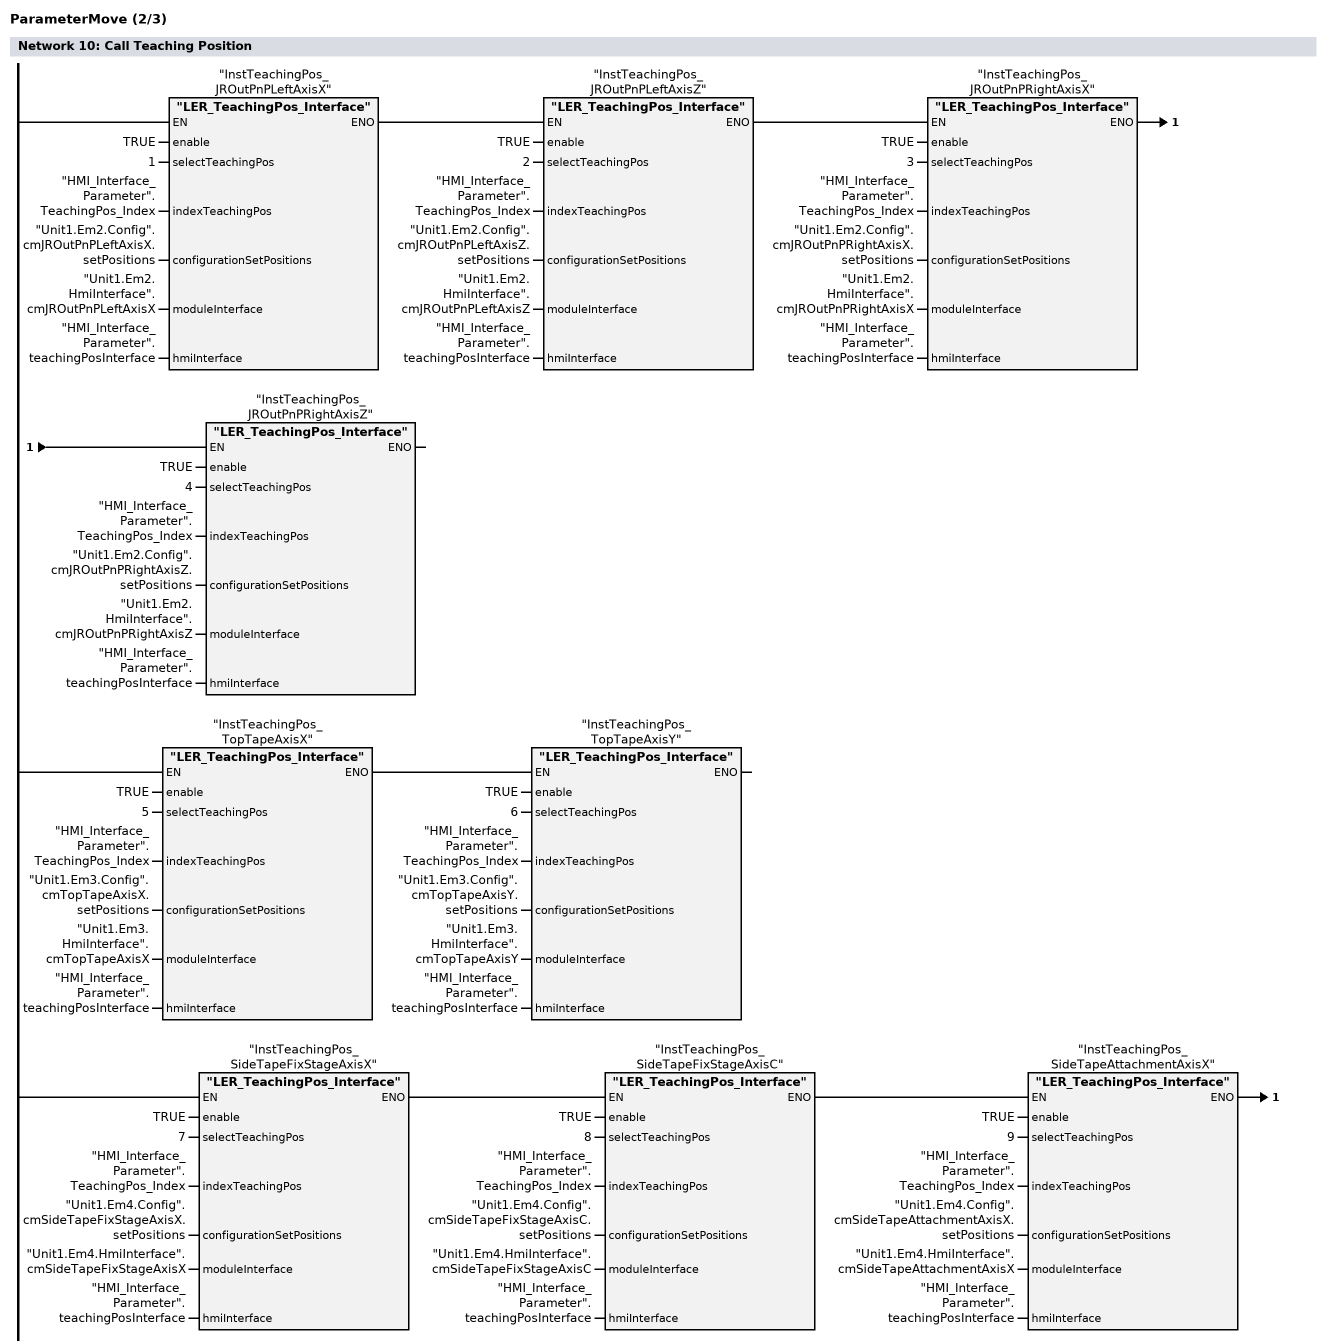
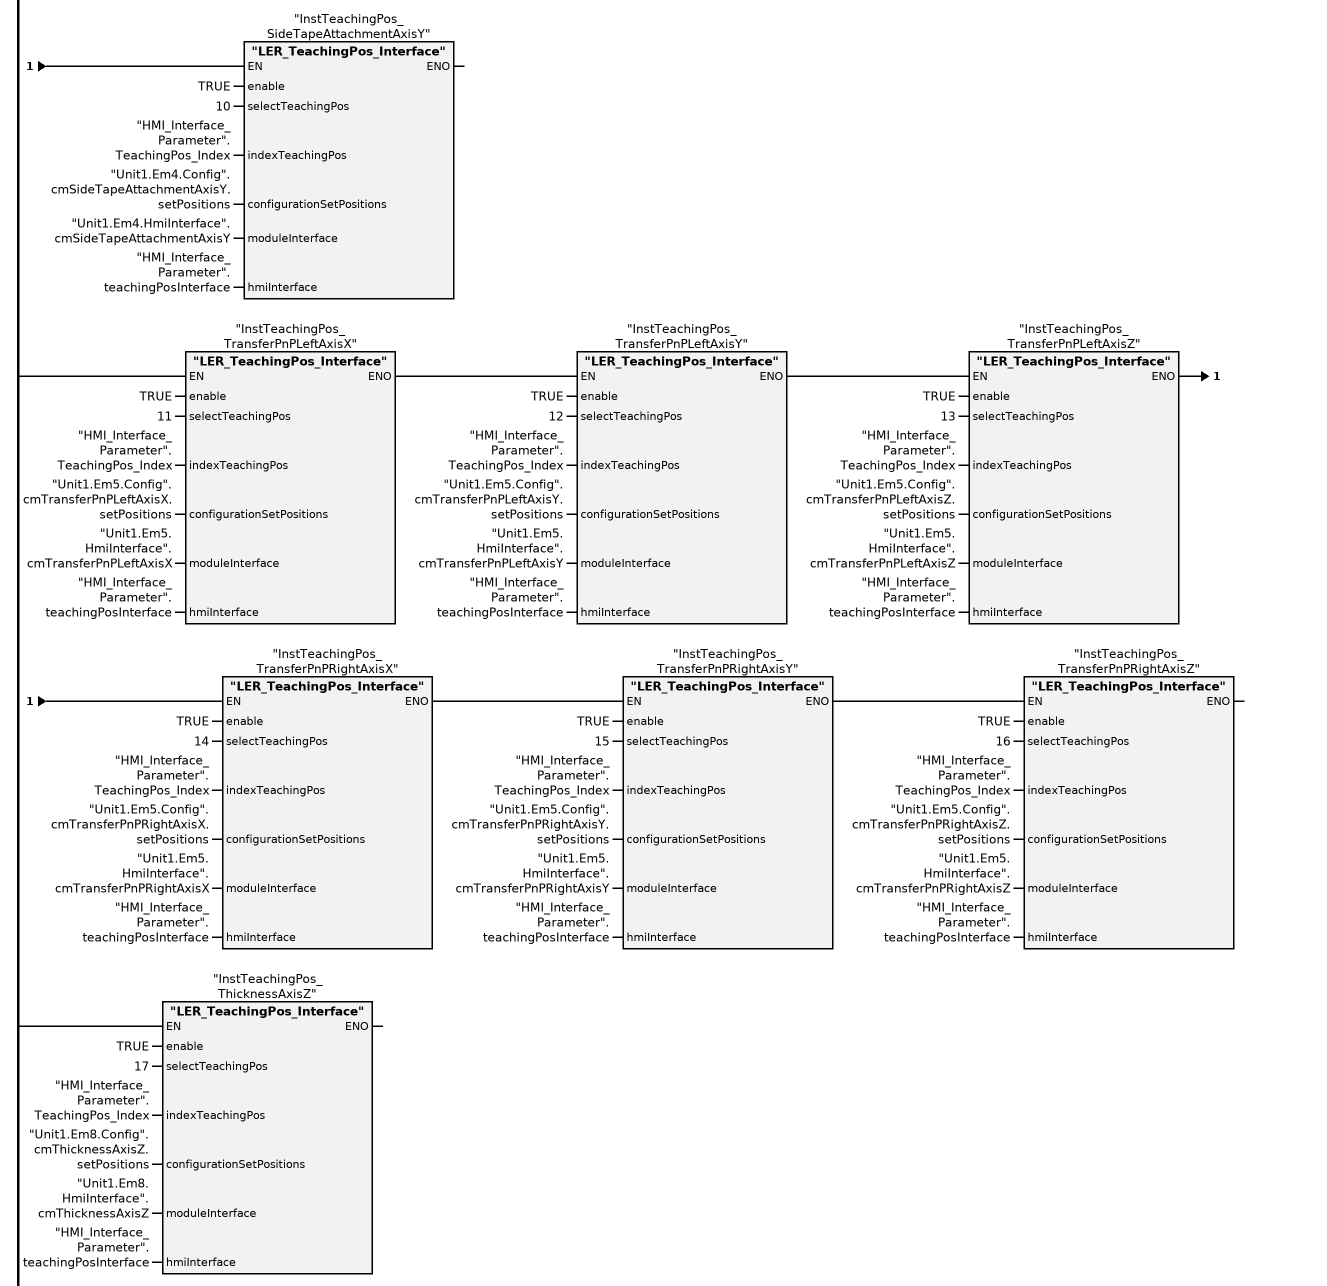
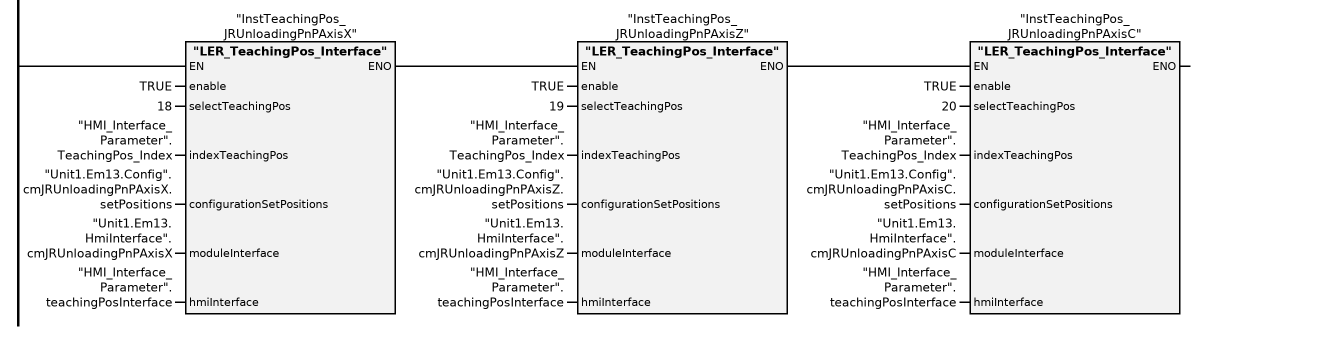
   RUNG wire#powerrail
      "InstTeachingPos_JROutPnPLeftAxisX"(enable := TRUE, selectTeachingPos := 1, indexTeachingPos := "HMI_Interface_Parameter".TeachingPos_Index, configurationSetPositions := "Unit1.Em2.Config".cmJROutPnPLeftAxisX.setPositions, moduleInterface := "Unit1.Em2.HmiInterface".cmJROutPnPLeftAxisX, hmiInterface := "HMI_Interface_Parameter".teachingPosInterface)
      "InstTeachingPos_JROutPnPLeftAxisZ"(enable := TRUE, selectTeachingPos := 2, indexTeachingPos := "HMI_Interface_Parameter".TeachingPos_Index, configurationSetPositions := "Unit1.Em2.Config".cmJROutPnPLeftAxisZ.setPositions, moduleInterface := "Unit1.Em2.HmiInterface".cmJROutPnPLeftAxisZ, hmiInterface := "HMI_Interface_Parameter".teachingPosInterface)
      "InstTeachingPos_JROutPnPRightAxisX"(enable := TRUE, selectTeachingPos := 3, indexTeachingPos := "HMI_Interface_Parameter".TeachingPos_Index, configurationSetPositions := "Unit1.Em2.Config".cmJROutPnPRightAxisX.setPositions, moduleInterface := "Unit1.Em2.HmiInterface".cmJROutPnPRightAxisX, hmiInterface := "HMI_Interface_Parameter".teachingPosInterface)
      "InstTeachingPos_JROutPnPRightAxisZ"(enable := TRUE, selectTeachingPos := 4, indexTeachingPos := "HMI_Interface_Parameter".TeachingPos_Index, configurationSetPositions := "Unit1.Em2.Config".cmJROutPnPRightAxisZ.setPositions, moduleInterface := "Unit1.Em2.HmiInterface".cmJROutPnPRightAxisZ, hmiInterface := "HMI_Interface_Parameter".teachingPosInterface)
   END_RUNG
   RUNG wire#powerrail
      "InstTeachingPos_TopTapeAxisX"(enable := TRUE, selectTeachingPos := 5, indexTeachingPos := "HMI_Interface_Parameter".TeachingPos_Index, configurationSetPositions := "Unit1.Em3.Config".cmTopTapeAxisX.setPositions, moduleInterface := "Unit1.Em3.HmiInterface".cmTopTapeAxisX, hmiInterface := "HMI_Interface_Parameter".teachingPosInterface)
      "InstTeachingPos_TopTapeAxisY"(enable := TRUE, selectTeachingPos := 6, indexTeachingPos := "HMI_Interface_Parameter".TeachingPos_Index, configurationSetPositions := "Unit1.Em3.Config".cmTopTapeAxisY.setPositions, moduleInterface := "Unit1.Em3.HmiInterface".cmTopTapeAxisY, hmiInterface := "HMI_Interface_Parameter".teachingPosInterface)
   END_RUNG
   RUNG wire#powerrail
      "InstTeachingPos_SideTapeFixStageAxisX"(enable := TRUE, selectTeachingPos := 7, indexTeachingPos := "HMI_Interface_Parameter".TeachingPos_Index, configurationSetPositions := "Unit1.Em4.Config".cmSideTapeFixStageAxisX.setPositions, moduleInterface := "Unit1.Em4.HmiInterface".cmSideTapeFixStageAxisX, hmiInterface := "HMI_Interface_Parameter".teachingPosInterface)
      "InstTeachingPos_SideTapeFixStageAxisC"(enable := TRUE, selectTeachingPos := 8, indexTeachingPos := "HMI_Interface_Parameter".TeachingPos_Index, configurationSetPositions := "Unit1.Em4.Config".cmSideTapeFixStageAxisC.setPositions, moduleInterface := "Unit1.Em4.HmiInterface".cmSideTapeFixStageAxisC, hmiInterface := "HMI_Interface_Parameter".teachingPosInterface)
      "InstTeachingPos_SideTapeAttachmentAxisX"(enable := TRUE, selectTeachingPos := 9, indexTeachingPos := "HMI_Interface_Parameter".TeachingPos_Index, configurationSetPositions := "Unit1.Em4.Config".cmSideTapeAttachmentAxisX.setPositions, moduleInterface := "Unit1.Em4.HmiInterface".cmSideTapeAttachmentAxisX, hmiInterface := "HMI_Interface_Parameter".teachingPosInterface)
      "InstTeachingPos_SideTapeAttachmentAxisY"(enable := TRUE, selectTeachingPos := 10, indexTeachingPos := "HMI_Interface_Parameter".TeachingPos_Index, configurationSetPositions := "Unit1.Em4.Config".cmSideTapeAttachmentAxisY.setPositions, moduleInterface := "Unit1.Em4.HmiInterface".cmSideTapeAttachmentAxisY, hmiInterface := "HMI_Interface_Parameter".teachingPosInterface)
   END_RUNG
   RUNG wire#powerrail
      "InstTeachingPos_TransferPnPLeftAxisX"(enable := TRUE, selectTeachingPos := 11, indexTeachingPos := "HMI_Interface_Parameter".TeachingPos_Index, configurationSetPositions := "Unit1.Em5.Config".cmTransferPnPLeftAxisX.setPositions, moduleInterface := "Unit1.Em5.HmiInterface".cmTransferPnPLeftAxisX, hmiInterface := "HMI_Interface_Parameter".teachingPosInterface)
      "InstTeachingPos_TransferPnPLeftAxisY"(enable := TRUE, selectTeachingPos := 12, indexTeachingPos := "HMI_Interface_Parameter".TeachingPos_Index, configurationSetPositions := "Unit1.Em5.Config".cmTransferPnPLeftAxisY.setPositions, moduleInterface := "Unit1.Em5.HmiInterface".cmTransferPnPLeftAxisY, hmiInterface := "HMI_Interface_Parameter".teachingPosInterface)
      "InstTeachingPos_TransferPnPLeftAxisZ"(enable := TRUE, selectTeachingPos := 13, indexTeachingPos := "HMI_Interface_Parameter".TeachingPos_Index, configurationSetPositions := "Unit1.Em5.Config".cmTransferPnPLeftAxisZ.setPositions, moduleInterface := "Unit1.Em5.HmiInterface".cmTransferPnPLeftAxisZ, hmiInterface := "HMI_Interface_Parameter".teachingPosInterface)
      "InstTeachingPos_TransferPnPRightAxisX"(enable := TRUE, selectTeachingPos := 14, indexTeachingPos := "HMI_Interface_Parameter".TeachingPos_Index, configurationSetPositions := "Unit1.Em5.Config".cmTransferPnPRightAxisX.setPositions, moduleInterface := "Unit1.Em5.HmiInterface".cmTransferPnPRightAxisX, hmiInterface := "HMI_Interface_Parameter".teachingPosInterface)
      "InstTeachingPos_TransferPnPRightAxisY"(enable := TRUE, selectTeachingPos := 15, indexTeachingPos := "HMI_Interface_Parameter".TeachingPos_Index, configurationSetPositions := "Unit1.Em5.Config".cmTransferPnPRightAxisY.setPositions, moduleInterface := "Unit1.Em5.HmiInterface".cmTransferPnPRightAxisY, hmiInterface := "HMI_Interface_Parameter".teachingPosInterface)
      "InstTeachingPos_TransferPnPRightAxisZ"(enable := TRUE, selectTeachingPos := 16, indexTeachingPos := "HMI_Interface_Parameter".TeachingPos_Index, configurationSetPositions := "Unit1.Em5.Config".cmTransferPnPRightAxisZ.setPositions, moduleInterface := "Unit1.Em5.HmiInterface".cmTransferPnPRightAxisZ, hmiInterface := "HMI_Interface_Parameter".teachingPosInterface)
   END_RUNG
   RUNG wire#powerrail
      "InstTeachingPos_ThicknessAxisZ"(enable := TRUE, selectTeachingPos := 17, indexTeachingPos := "HMI_Interface_Parameter".TeachingPos_Index, configurationSetPositions := "Unit1.Em8.Config".cmThicknessAxisZ.setPositions, moduleInterface := "Unit1.Em8.HmiInterface".cmThicknessAxisZ, hmiInterface := "HMI_Interface_Parameter".teachingPosInterface)
   END_RUNG
   RUNG wire#powerrail
      "InstTeachingPos_JRUnloadingPnPAxisX"(enable := TRUE, selectTeachingPos := 18, indexTeachingPos := "HMI_Interface_Parameter".TeachingPos_Index, configurationSetPositions := "Unit1.Em13.Config".cmJRUnloadingPnPAxisX.setPositions, moduleInterface := "Unit1.Em13.HmiInterface".cmJRUnloadingPnPAxisX, hmiInterface := "HMI_Interface_Parameter".teachingPosInterface)
      "InstTeachingPos_JRUnloadingPnPAxisZ"(enable := TRUE, selectTeachingPos := 19, indexTeachingPos := "HMI_Interface_Parameter".TeachingPos_Index, configurationSetPositions := "Unit1.Em13.Config".cmJRUnloadingPnPAxisZ.setPositions, moduleInterface := "Unit1.Em13.HmiInterface".cmJRUnloadingPnPAxisZ, hmiInterface := "HMI_Interface_Parameter".teachingPosInterface)
      "InstTeachingPos_JRUnloadingPnPAxisC"(enable := TRUE, selectTeachingPos := 20, indexTeachingPos := "HMI_Interface_Parameter".TeachingPos_Index, configurationSetPositions := "Unit1.Em13.Config".cmJRUnloadingPnPAxisC.setPositions, moduleInterface := "Unit1.Em13.HmiInterface".cmJRUnloadingPnPAxisC, hmiInterface := "HMI_Interface_Parameter".teachingPosInterface)
   END_RUNG
   // the same network as SCL:
   "InstTeachingPos_JROutPnPLeftAxisX"(enable := TRUE,   // "LER_TeachingPos_Interface"
                           selectTeachingPos := 1,
                           indexTeachingPos := "HMI_Interface_Parameter".TeachingPos_Index,
                           configurationSetPositions := "Unit1.Em2.Config".cmJROutPnPLeftAxisX.setPositions,
                           moduleInterface := "Unit1.Em2.HmiInterface".cmJROutPnPLeftAxisX,
                           hmiInterface := "HMI_Interface_Parameter".teachingPosInterface,
                           ENO => #_w1);
   "InstTeachingPos_JROutPnPLeftAxisZ"(EN := #_w1,   // "LER_TeachingPos_Interface"
                           enable := TRUE,
                           selectTeachingPos := 2,
                           indexTeachingPos := "HMI_Interface_Parameter".TeachingPos_Index,
                           configurationSetPositions := "Unit1.Em2.Config".cmJROutPnPLeftAxisZ.setPositions,
                           moduleInterface := "Unit1.Em2.HmiInterface".cmJROutPnPLeftAxisZ,
                           hmiInterface := "HMI_Interface_Parameter".teachingPosInterface,
                           ENO => #_w2);
   "InstTeachingPos_JROutPnPRightAxisX"(EN := #_w2,   // "LER_TeachingPos_Interface"
                           enable := TRUE,
                           selectTeachingPos := 3,
                           indexTeachingPos := "HMI_Interface_Parameter".TeachingPos_Index,
                           configurationSetPositions := "Unit1.Em2.Config".cmJROutPnPRightAxisX.setPositions,
                           moduleInterface := "Unit1.Em2.HmiInterface".cmJROutPnPRightAxisX,
                           hmiInterface := "HMI_Interface_Parameter".teachingPosInterface,
                           ENO => #_w3);
   IF #_w3 THEN
       "InstTeachingPos_JROutPnPRightAxisZ"(enable := TRUE,   // "LER_TeachingPos_Interface"
                               selectTeachingPos := 4,
                               indexTeachingPos := "HMI_Interface_Parameter".TeachingPos_Index,
                               configurationSetPositions := "Unit1.Em2.Config".cmJROutPnPRightAxisZ.setPositions,
                               moduleInterface := "Unit1.Em2.HmiInterface".cmJROutPnPRightAxisZ,
                               hmiInterface := "HMI_Interface_Parameter".teachingPosInterface);
   END_IF;
   "InstTeachingPos_TopTapeAxisX"(enable := TRUE,   // "LER_TeachingPos_Interface"
                           selectTeachingPos := 5,
                           indexTeachingPos := "HMI_Interface_Parameter".TeachingPos_Index,
                           configurationSetPositions := "Unit1.Em3.Config".cmTopTapeAxisX.setPositions,
                           moduleInterface := "Unit1.Em3.HmiInterface".cmTopTapeAxisX,
                           hmiInterface := "HMI_Interface_Parameter".teachingPosInterface,
                           ENO => #_w4);
   IF #_w4 THEN
       "InstTeachingPos_TopTapeAxisY"(enable := TRUE,   // "LER_TeachingPos_Interface"
                               selectTeachingPos := 6,
                               indexTeachingPos := "HMI_Interface_Parameter".TeachingPos_Index,
                               configurationSetPositions := "Unit1.Em3.Config".cmTopTapeAxisY.setPositions,
                               moduleInterface := "Unit1.Em3.HmiInterface".cmTopTapeAxisY,
                               hmiInterface := "HMI_Interface_Parameter".teachingPosInterface);
   END_IF;
   "InstTeachingPos_SideTapeFixStageAxisX"(enable := TRUE,   // "LER_TeachingPos_Interface"
                           selectTeachingPos := 7,
                           indexTeachingPos := "HMI_Interface_Parameter".TeachingPos_Index,
                           configurationSetPositions := "Unit1.Em4.Config".cmSideTapeFixStageAxisX.setPositions,
                           moduleInterface := "Unit1.Em4.HmiInterface".cmSideTapeFixStageAxisX,
                           hmiInterface := "HMI_Interface_Parameter".teachingPosInterface,
                           ENO => #_w5);
   "InstTeachingPos_SideTapeFixStageAxisC"(EN := #_w5,   // "LER_TeachingPos_Interface"
                           enable := TRUE,
                           selectTeachingPos := 8,
                           indexTeachingPos := "HMI_Interface_Parameter".TeachingPos_Index,
                           configurationSetPositions := "Unit1.Em4.Config".cmSideTapeFixStageAxisC.setPositions,
                           moduleInterface := "Unit1.Em4.HmiInterface".cmSideTapeFixStageAxisC,
                           hmiInterface := "HMI_Interface_Parameter".teachingPosInterface,
                           ENO => #_w6);
   "InstTeachingPos_SideTapeAttachmentAxisX"(EN := #_w6,   // "LER_TeachingPos_Interface"
                           enable := TRUE,
                           selectTeachingPos := 9,
                           indexTeachingPos := "HMI_Interface_Parameter".TeachingPos_Index,
                           configurationSetPositions := "Unit1.Em4.Config".cmSideTapeAttachmentAxisX.setPositions,
                           moduleInterface := "Unit1.Em4.HmiInterface".cmSideTapeAttachmentAxisX,
                           hmiInterface := "HMI_Interface_Parameter".teachingPosInterface,
                           ENO => #_w7);
   IF #_w7 THEN
       "InstTeachingPos_SideTapeAttachmentAxisY"(enable := TRUE,   // "LER_TeachingPos_Interface"
                               selectTeachingPos := 10,
                               indexTeachingPos := "HMI_Interface_Parameter".TeachingPos_Index,
                               configurationSetPositions := "Unit1.Em4.Config".cmSideTapeAttachmentAxisY.setPositions,
                               moduleInterface := "Unit1.Em4.HmiInterface".cmSideTapeAttachmentAxisY,
                               hmiInterface := "HMI_Interface_Parameter".teachingPosInterface);
   END_IF;
   "InstTeachingPos_TransferPnPLeftAxisX"(enable := TRUE,   // "LER_TeachingPos_Interface"
                           selectTeachingPos := 11,
                           indexTeachingPos := "HMI_Interface_Parameter".TeachingPos_Index,
                           configurationSetPositions := "Unit1.Em5.Config".cmTransferPnPLeftAxisX.setPositions,
                           moduleInterface := "Unit1.Em5.HmiInterface".cmTransferPnPLeftAxisX,
                           hmiInterface := "HMI_Interface_Parameter".teachingPosInterface,
                           ENO => #_w8);
   "InstTeachingPos_TransferPnPLeftAxisY"(EN := #_w8,   // "LER_TeachingPos_Interface"
                           enable := TRUE,
                           selectTeachingPos := 12,
                           indexTeachingPos := "HMI_Interface_Parameter".TeachingPos_Index,
                           configurationSetPositions := "Unit1.Em5.Config".cmTransferPnPLeftAxisY.setPositions,
                           moduleInterface := "Unit1.Em5.HmiInterface".cmTransferPnPLeftAxisY,
                           hmiInterface := "HMI_Interface_Parameter".teachingPosInterface,
                           ENO => #_w9);
   "InstTeachingPos_TransferPnPLeftAxisZ"(EN := #_w9,   // "LER_TeachingPos_Interface"
                           enable := TRUE,
                           selectTeachingPos := 13,
                           indexTeachingPos := "HMI_Interface_Parameter".TeachingPos_Index,
                           configurationSetPositions := "Unit1.Em5.Config".cmTransferPnPLeftAxisZ.setPositions,
                           moduleInterface := "Unit1.Em5.HmiInterface".cmTransferPnPLeftAxisZ,
                           hmiInterface := "HMI_Interface_Parameter".teachingPosInterface,
                           ENO => #_w10);
   "InstTeachingPos_TransferPnPRightAxisX"(EN := #_w10,   // "LER_TeachingPos_Interface"
                           enable := TRUE,
                           selectTeachingPos := 14,
                           indexTeachingPos := "HMI_Interface_Parameter".TeachingPos_Index,
                           configurationSetPositions := "Unit1.Em5.Config".cmTransferPnPRightAxisX.setPositions,
                           moduleInterface := "Unit1.Em5.HmiInterface".cmTransferPnPRightAxisX,
                           hmiInterface := "HMI_Interface_Parameter".teachingPosInterface,
                           ENO => #_w11);
   "InstTeachingPos_TransferPnPRightAxisY"(EN := #_w11,   // "LER_TeachingPos_Interface"
                           enable := TRUE,
                           selectTeachingPos := 15,
                           indexTeachingPos := "HMI_Interface_Parameter".TeachingPos_Index,
                           configurationSetPositions := "Unit1.Em5.Config".cmTransferPnPRightAxisY.setPositions,
                           moduleInterface := "Unit1.Em5.HmiInterface".cmTransferPnPRightAxisY,
                           hmiInterface := "HMI_Interface_Parameter".teachingPosInterface,
                           ENO => #_w12);
   IF #_w12 THEN
       "InstTeachingPos_TransferPnPRightAxisZ"(enable := TRUE,   // "LER_TeachingPos_Interface"
                               selectTeachingPos := 16,
                               indexTeachingPos := "HMI_Interface_Parameter".TeachingPos_Index,
                               configurationSetPositions := "Unit1.Em5.Config".cmTransferPnPRightAxisZ.setPositions,
                               moduleInterface := "Unit1.Em5.HmiInterface".cmTransferPnPRightAxisZ,
                               hmiInterface := "HMI_Interface_Parameter".teachingPosInterface);
   END_IF;
   "InstTeachingPos_ThicknessAxisZ"(enable := TRUE,   // "LER_TeachingPos_Interface"
                           selectTeachingPos := 17,
                           indexTeachingPos := "HMI_Interface_Parameter".TeachingPos_Index,
                           configurationSetPositions := "Unit1.Em8.Config".cmThicknessAxisZ.setPositions,
                           moduleInterface := "Unit1.Em8.HmiInterface".cmThicknessAxisZ,
                           hmiInterface := "HMI_Interface_Parameter".teachingPosInterface);
   "InstTeachingPos_JRUnloadingPnPAxisX"(enable := TRUE,   // "LER_TeachingPos_Interface"
                           selectTeachingPos := 18,
                           indexTeachingPos := "HMI_Interface_Parameter".TeachingPos_Index,
                           configurationSetPositions := "Unit1.Em13.Config".cmJRUnloadingPnPAxisX.setPositions,
                           moduleInterface := "Unit1.Em13.HmiInterface".cmJRUnloadingPnPAxisX,
                           hmiInterface := "HMI_Interface_Parameter".teachingPosInterface,
                           ENO => #_w13);
   "InstTeachingPos_JRUnloadingPnPAxisZ"(EN := #_w13,   // "LER_TeachingPos_Interface"
                           enable := TRUE,
                           selectTeachingPos := 19,
                           indexTeachingPos := "HMI_Interface_Parameter".TeachingPos_Index,
                           configurationSetPositions := "Unit1.Em13.Config".cmJRUnloadingPnPAxisZ.setPositions,
                           moduleInterface := "Unit1.Em13.HmiInterface".cmJRUnloadingPnPAxisZ,
                           hmiInterface := "HMI_Interface_Parameter".teachingPosInterface,
                           ENO => #_w14);
   IF #_w14 THEN
       "InstTeachingPos_JRUnloadingPnPAxisC"(enable := TRUE,   // "LER_TeachingPos_Interface"
                               selectTeachingPos := 20,
                               indexTeachingPos := "HMI_Interface_Parameter".TeachingPos_Index,
                               configurationSetPositions := "Unit1.Em13.Config".cmJRUnloadingPnPAxisC.setPositions,
                               moduleInterface := "Unit1.Em13.HmiInterface".cmJRUnloadingPnPAxisC,
                               hmiInterface := "HMI_Interface_Parameter".teachingPosInterface);
   END_IF;
END_REGION

REGION Network 11: Call Distance
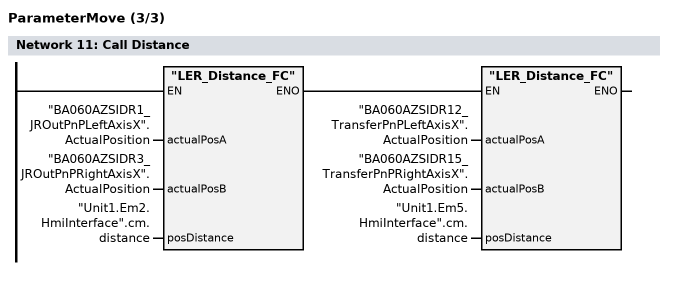
   RUNG wire#powerrail
      "LER_Distance_FC"(actualPosA := "BA060AZSIDR1_JROutPnPLeftAxisX".ActualPosition, actualPosB := "BA060AZSIDR3_JROutPnPRightAxisX".ActualPosition, posDistance := "Unit1.Em2.HmiInterface".cm.distance)
      "LER_Distance_FC"(actualPosA := "BA060AZSIDR12_TransferPnPLeftAxisX".ActualPosition, actualPosB := "BA060AZSIDR15_TransferPnPRightAxisX".ActualPosition, posDistance := "Unit1.Em5.HmiInterface".cm.distance)
   END_RUNG
   // the same network as SCL:
   "LER_Distance_FC"(actualPosA := "BA060AZSIDR1_JROutPnPLeftAxisX".ActualPosition,
                     actualPosB := "BA060AZSIDR3_JROutPnPRightAxisX".ActualPosition,
                     posDistance := "Unit1.Em2.HmiInterface".cm.distance,
                     ENO => #_w1);
   IF #_w1 THEN
       "LER_Distance_FC"(actualPosA := "BA060AZSIDR12_TransferPnPLeftAxisX".ActualPosition,
                         actualPosB := "BA060AZSIDR15_TransferPnPRightAxisX".ActualPosition,
                         posDistance := "Unit1.Em5.HmiInterface".cm.distance);
   END_IF;
END_REGION
END_FUNCTION

FUNCTION "PrameterMove_Legacy" : Void
{ S7_Optimized_Access := 'TRUE' ; Published := 'FALSE' }
VERSION : 0.1
   VAR_TEMP 
      tempIndex : Int;
   END_VAR


BEGIN
	REGION PLC → HMI
	    
	    // Recipe
	    // IF "HMI_Interface_Parameter".RecipeButton.Read THEN
	    //      "RecipeParameter".currentRecipeName := Unit1.EmNodes.unitRecipe.currentRecipeName;
	    //      "RecipeParameter".currentRecipeID := Unit1.EmNodes.unitRecipe.currentRecipeID;
	    //     "RecipeParameter".unitRecipe := Unit1.EmNodes.unitRecipe.unitRecipe;
	       
	    // END_IF;
	    
	    // FAT Parameter
	(*    "HMI_Interface_Parameter".FATModeInterface.HoursTest.ProcessValue.ProcTimeLeft := Unit1.EmNodes.FATModeInterface.HoursTest.ProcessValue.ProcTimeLeft;
	    "HMI_Interface_Parameter".FATModeInterface.Capability.ProcessValue.CapabilityCount := Unit1.EmNodes.FATModeInterface.Capability.ProcessValue.CapabilityCount;
	    "HMI_Interface_Parameter".FATModeInterface.Sampling.ProcessValue.CellCount := Unit1.EmNodes.FATModeInterface.Sampling.ProcessValue.CellCount; *)
	    
	    Unit1.EmNodes.FATModeInterface.HoursTest.SetValue.SelectHours_SetValue := "HMI_Interface_Parameter".FATModeInterface.HoursTest.SetValue.SelectHours_SetValue;
	    Unit1.EmNodes.FATModeInterface.Capability.SetValue.SelectCycle_SetValue := "HMI_Interface_Parameter".FATModeInterface.Capability.SetValue.SelectCycle_SetValue;
	    Unit1.EmNodes.FATModeInterface.Sampling.SetValue.SelectCount_SetValue := "HMI_Interface_Parameter".FATModeInterface.Sampling.SetValue.SelectCount_SetValue;
	    
	(*    "HMI_Interface_Parameter".FATModeInterface.HoursTest.ProcessValue.SelectHours_ProcessValue := Unit1.EmNodes.FATModeInterface.HoursTest.ProcessValue.SelectHours_ProcessValue;
	    "HMI_Interface_Parameter".FATModeInterface.Capability.ProcessValue.SelectCycle_ProcessValue := Unit1.EmNodes.FATModeInterface.Capability.ProcessValue.SelectCycle_ProcessValue;
	    "HMI_Interface_Parameter".FATModeInterface.Sampling.ProcessValue.SelectCount_ProcessValue := Unit1.EmNodes.FATModeInterface.Sampling.ProcessValue.SelectCount_ProcessValue; *)
	END_REGION
	
	REGION HMI → PLC
	    
	    // Select equipment
	    // Unit1.EmNodes.unitRecipe.processUnitNo := "HMI_Interface_Parameter".ProcessUnitSelect;
	    // Unit1.EmNodes.unitRecipe.selectedRecipeTypeID := "RecipeParameter".selectedRecipeTypeID;
	    // Unit1.EmNodes.unitRecipe.selectedRecipeID := "RecipeParameter".selectedRecipeID;
	    
	    // Recipe
	    //IF "HMI_Interface_Parameter".RecipeButton.Apply THEN
	(*        // Unit1.EmNodes.unitRecipe.currentRecipeName := "RecipeParameter".currentRecipeName;
	        // Unit1.EmNodes.unitRecipe.currentRecipeID := "RecipeParameter".currentRecipeID;
	        //Unit1.EmNodes.unitRecipe.unitRecipe := "RecipeParameter".unitRecipe;
	        
	        //이 외 레시피는 Program(SV,PV 비교) 및 UDT 수정 필요.
	        
	        // Parameter
	        //Unit or Em parameter := "HMI_Interface_Parameter".Distance[1]."Process Value" := "HMI_Interface_Parameter".Distance[1]."Set Value";
	        //...
	        
	        
	        // FAT SV -> PV
	        
	        Unit1.EmNodes.FATModeInterface.HoursTest.ProcessValue.SelectHours_ProcessValue := Unit1.EmNodes.FATModeInterface.HoursTest.SetValue.SelectHours_SetValue;
	        Unit1.EmNodes.FATModeInterface.Capability.ProcessValue.SelectCycle_ProcessValue := Unit1.EmNodes.FATModeInterface.Capability.SetValue.SelectCycle_SetValue;
	        Unit1.EmNodes.FATModeInterface.Sampling.ProcessValue.SelectCount_ProcessValue := Unit1.EmNodes.FATModeInterface.Sampling.SetValue.SelectCount_SetValue; *)
	    //END_IF;
	    
	    // FAT Parameter
	(*    Unit1.EmNodes.FATModeSelect.HoursTestMode := "HMI_Interface_Parameter".FATModeSelect.HoursTestMode;
	    Unit1.EmNodes.FATModeSelect.CapabilityMode := "HMI_Interface_Parameter".FATModeSelect.CapabilityMode;
	    Unit1.EmNodes.FATModeSelect.SamplingMode := "HMI_Interface_Parameter".FATModeSelect.SamplingMode; *)
	    
	END_REGION
END_FUNCTION

FUNCTION "CallSimulation" : Void   // FC22, LAD
TITLE = CallSimulation
// This blocks switches between simulation with SIMIT and PLCSIM Advanced or with PLCSIM and PLC internal simulation function blocks
// stored: IsIECCheckEnabled true, SetENOAutomatically true
BEGIN
END_FUNCTION

FUNCTION "CallManualOperationLines_Unit1" : Void   // FC80, LAD
// stored: SetENOAutomatically false
   VAR_TEMP
      StatusEm : Array[0..13] of Struct
         Status : Array[0..40] of Word;
      END_STRUCT;
      errorIDEm : Array[0..13] of Struct
         errorID : Array[0..40] of Word;
      END_STRUCT;
      disableUnit1 : Bool;
      TempAxisCommands : "LBC_typeAxis64PosManualCommands";
      TempAxisMonitoring : "LBC_typeAxis64PosProcessValues";
      TempSoftCam : Array[0..8] of "LER_typeSoftCamParameter";
   END_VAR
   VAR CONSTANT
      MECHANIC_NAME_ENABLE : Bool;
   END_VAR
   VAR_TEMP   // added for the SCL form of the ladder/FBD networks
      _w1 : Bool;
   END_VAR
BEGIN

REGION Network 1: Unit 1 Enable Manual Operation
   // Condition to disable manual operation lines in Unit 3
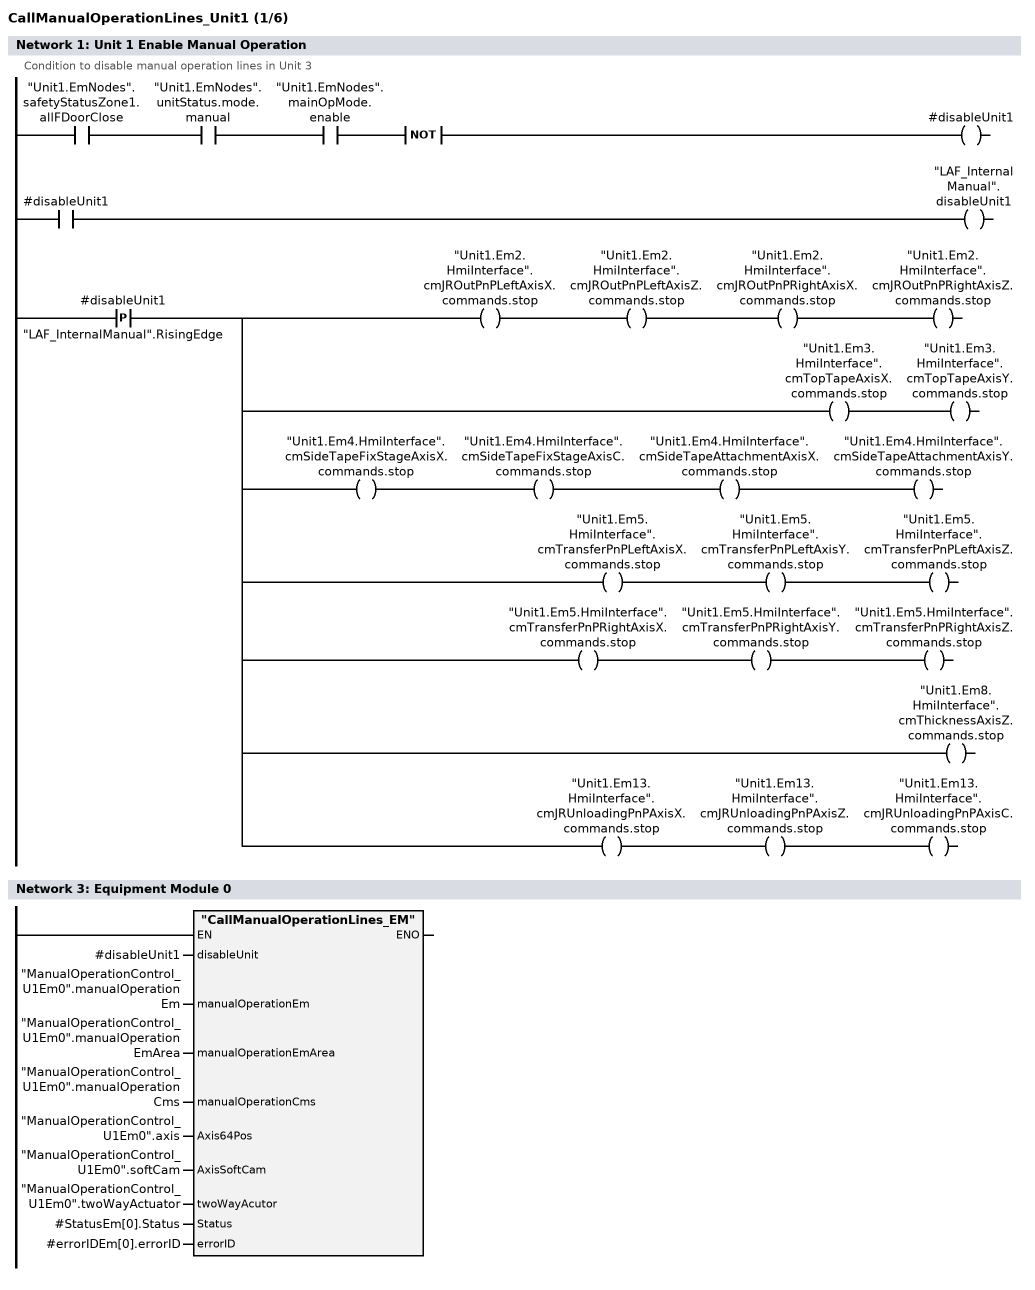
   RUNG wire#powerrail
      Contact( "Unit1.EmNodes".safetyStatusZone1.allFDoorClose )
      Contact( "Unit1.EmNodes".unitStatus.mode.manual )
      Contact( "Unit1.EmNodes".mainOpMode.enable )
      Not()
      Coil( #disableUnit1 )
   END_RUNG
   RUNG wire#powerrail
      Contact( #disableUnit1 )
      Coil( "LAF_InternalManual".disableUnit1 )
   END_RUNG
   RUNG wire#powerrail
      P_Contact(operand := #disableUnit1, bit := "LAF_InternalManual".RisingEdge)
      wire#w1
      Coil( "Unit1.Em2.HmiInterface".cmJROutPnPLeftAxisX.commands.stop )
      Coil( "Unit1.Em2.HmiInterface".cmJROutPnPLeftAxisZ.commands.stop )
      Coil( "Unit1.Em2.HmiInterface".cmJROutPnPRightAxisX.commands.stop )
      Coil( "Unit1.Em2.HmiInterface".cmJROutPnPRightAxisZ.commands.stop )
   END_RUNG
   RUNG wire#w1
      Coil( "Unit1.Em3.HmiInterface".cmTopTapeAxisX.commands.stop )
      Coil( "Unit1.Em3.HmiInterface".cmTopTapeAxisY.commands.stop )
   END_RUNG
   RUNG wire#w1
      Coil( "Unit1.Em4.HmiInterface".cmSideTapeFixStageAxisX.commands.stop )
      Coil( "Unit1.Em4.HmiInterface".cmSideTapeFixStageAxisC.commands.stop )
      Coil( "Unit1.Em4.HmiInterface".cmSideTapeAttachmentAxisX.commands.stop )
      Coil( "Unit1.Em4.HmiInterface".cmSideTapeAttachmentAxisY.commands.stop )
   END_RUNG
   RUNG wire#w1
      Coil( "Unit1.Em5.HmiInterface".cmTransferPnPLeftAxisX.commands.stop )
      Coil( "Unit1.Em5.HmiInterface".cmTransferPnPLeftAxisY.commands.stop )
      Coil( "Unit1.Em5.HmiInterface".cmTransferPnPLeftAxisZ.commands.stop )
   END_RUNG
   RUNG wire#w1
      Coil( "Unit1.Em5.HmiInterface".cmTransferPnPRightAxisX.commands.stop )
      Coil( "Unit1.Em5.HmiInterface".cmTransferPnPRightAxisY.commands.stop )
      Coil( "Unit1.Em5.HmiInterface".cmTransferPnPRightAxisZ.commands.stop )
   END_RUNG
   RUNG wire#w1
      Coil( "Unit1.Em8.HmiInterface".cmThicknessAxisZ.commands.stop )
   END_RUNG
   RUNG wire#w1
      Coil( "Unit1.Em13.HmiInterface".cmJRUnloadingPnPAxisX.commands.stop )
      Coil( "Unit1.Em13.HmiInterface".cmJRUnloadingPnPAxisZ.commands.stop )
      Coil( "Unit1.Em13.HmiInterface".cmJRUnloadingPnPAxisC.commands.stop )
   END_RUNG
   // the same network as SCL:
   #disableUnit1 := NOT ("Unit1.EmNodes".safetyStatusZone1.allFDoorClose AND "Unit1.EmNodes".unitStatus.mode.manual AND "Unit1.EmNodes".mainOpMode.enable);
   "LAF_InternalManual".disableUnit1 := #disableUnit1;
   #_w1 := #disableUnit1 AND NOT "LAF_InternalManual".RisingEdge;   // rising edge of #disableUnit1
   "LAF_InternalManual".RisingEdge := #disableUnit1;
   "Unit1.Em2.HmiInterface".cmJROutPnPLeftAxisX.commands.stop := #_w1;
   "Unit1.Em2.HmiInterface".cmJROutPnPLeftAxisZ.commands.stop := #_w1;
   "Unit1.Em2.HmiInterface".cmJROutPnPRightAxisX.commands.stop := #_w1;
   "Unit1.Em2.HmiInterface".cmJROutPnPRightAxisZ.commands.stop := #_w1;
   "Unit1.Em3.HmiInterface".cmTopTapeAxisX.commands.stop := #_w1;
   "Unit1.Em3.HmiInterface".cmTopTapeAxisY.commands.stop := #_w1;
   "Unit1.Em4.HmiInterface".cmSideTapeFixStageAxisX.commands.stop := #_w1;
   "Unit1.Em4.HmiInterface".cmSideTapeFixStageAxisC.commands.stop := #_w1;
   "Unit1.Em4.HmiInterface".cmSideTapeAttachmentAxisX.commands.stop := #_w1;
   "Unit1.Em4.HmiInterface".cmSideTapeAttachmentAxisY.commands.stop := #_w1;
   "Unit1.Em5.HmiInterface".cmTransferPnPLeftAxisX.commands.stop := #_w1;
   "Unit1.Em5.HmiInterface".cmTransferPnPLeftAxisY.commands.stop := #_w1;
   "Unit1.Em5.HmiInterface".cmTransferPnPLeftAxisZ.commands.stop := #_w1;
   "Unit1.Em5.HmiInterface".cmTransferPnPRightAxisX.commands.stop := #_w1;
   "Unit1.Em5.HmiInterface".cmTransferPnPRightAxisY.commands.stop := #_w1;
   "Unit1.Em5.HmiInterface".cmTransferPnPRightAxisZ.commands.stop := #_w1;
   "Unit1.Em8.HmiInterface".cmThicknessAxisZ.commands.stop := #_w1;
   "Unit1.Em13.HmiInterface".cmJRUnloadingPnPAxisX.commands.stop := #_w1;
   "Unit1.Em13.HmiInterface".cmJRUnloadingPnPAxisZ.commands.stop := #_w1;
   "Unit1.Em13.HmiInterface".cmJRUnloadingPnPAxisC.commands.stop := #_w1;
END_REGION

REGION Network 2 (SCL): Equipment Module 0 Cms Mapping
   REGION Input Mapping
       // TwoWayActuator
       "ManualOperationControl_U1Em0".twoWayActuator[1].monitoring := "Unit1.Em0.HmiInterface".cmStacker1NgBoxClampMoverOpenClose.monitoring;
       "ManualOperationControl_U1Em0".twoWayActuator[2].monitoring := "Unit1.Em0.HmiInterface".cmStacker1NgBoxClampLeftOpenClose.monitoring;
       "ManualOperationControl_U1Em0".twoWayActuator[3].monitoring := "Unit1.Em0.HmiInterface".cmStacker1NgBoxClampRightOpenClose.monitoring;
       "ManualOperationControl_U1Em0".twoWayActuator[4].monitoring := "Unit1.Em0.HmiInterface".cmStacker1NgBoxLoadingUpDown.monitoring;
       "ManualOperationControl_U1Em0".twoWayActuator[5].monitoring := "Unit1.Em0.HmiInterface".cmStacker1NgBoxUnitMoverBwdFwd.monitoring;
       "ManualOperationControl_U1Em0".twoWayActuator[6].monitoring := "Unit1.Em0.HmiInterface".cmStacker1NgBoxLiftDownUp.monitoring;
       "ManualOperationControl_U1Em0".twoWayActuator[7].monitoring := "Unit1.Em0.HmiInterface".cmStacker1NgBoxLockDownUp.monitoring;
   END_REGION


